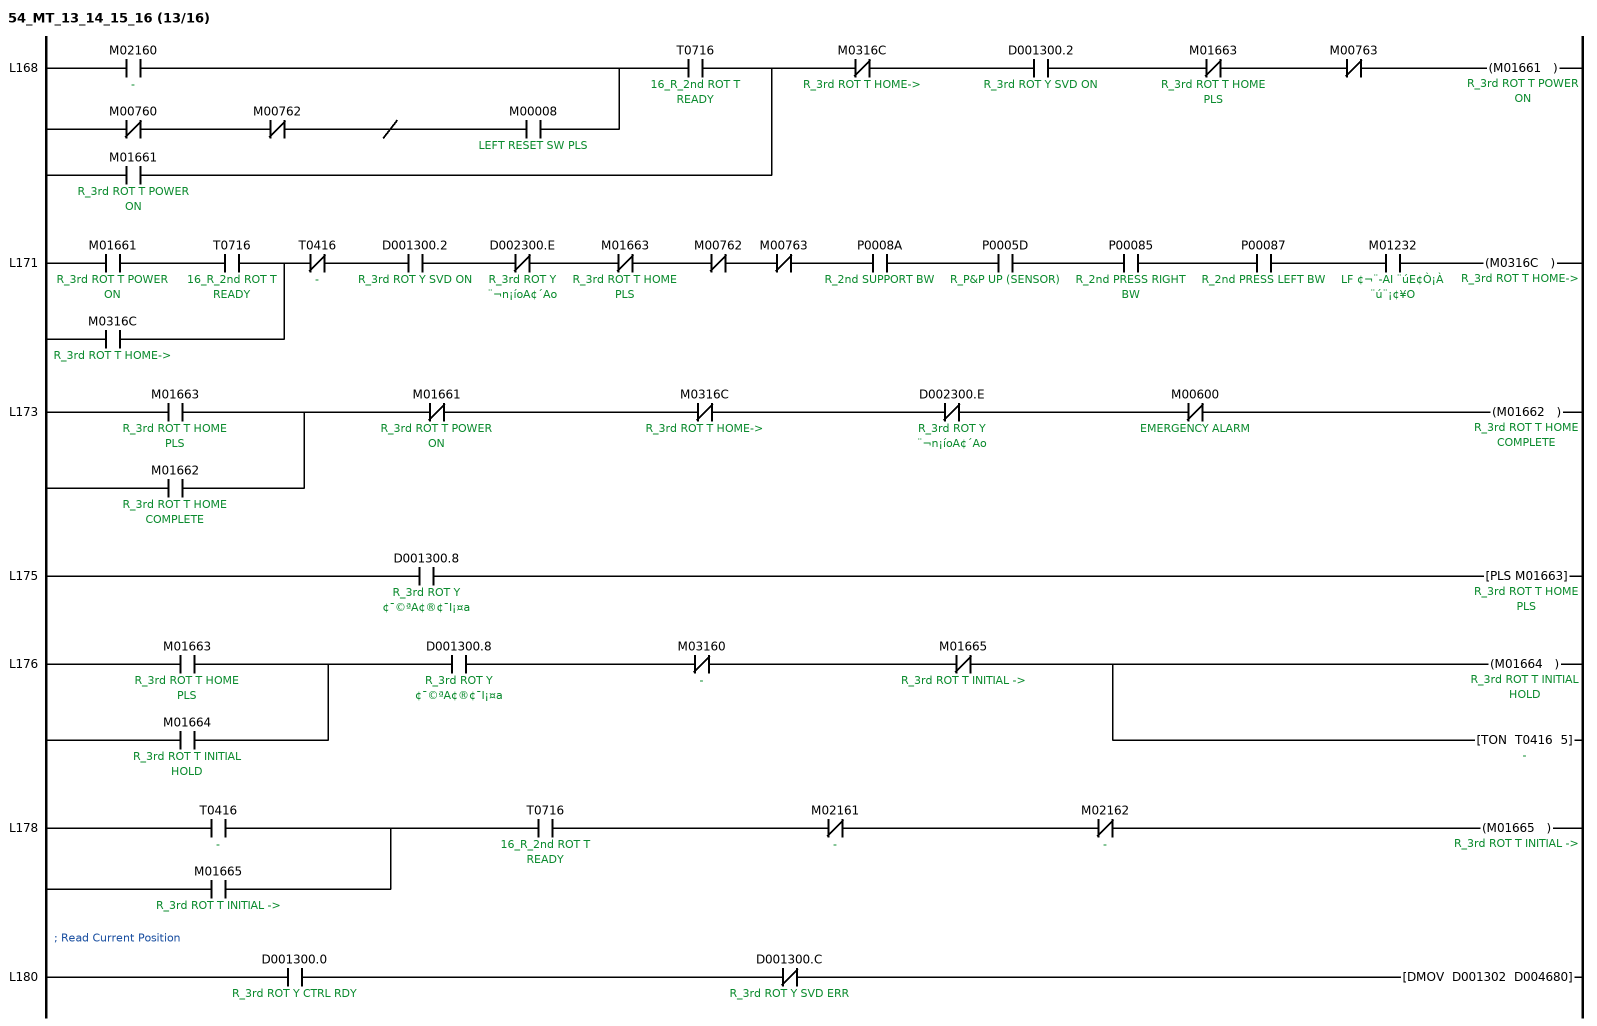
[picture p312: 54_MT_13_14_15_16 rungs L168-L180]
; L168
LOAD      M02160	// -
LOAD NOT  M00760
AND NOT   M00762
NOT
AND       M00008	// LEFT RESET SW PLS
OR LOAD
AND       T0716	// 16_R_2nd ROT T READY
OR        M01661	// R_3rd ROT T POWER ON
AND NOT   M0316C	// R_3rd ROT T HOME->
AND       D001300.2	// R_3rd ROT Y SVD ON
AND NOT   M01663	// R_3rd ROT T HOME PLS
AND NOT   M00763
OUT       M01661	// R_3rd ROT T POWER ON
; L171
LOAD      M01661	// R_3rd ROT T POWER ON
AND       T0716	// 16_R_2nd ROT T READY
OR        M0316C	// R_3rd ROT T HOME->
AND NOT   T0416	// -
AND       D001300.2	// R_3rd ROT Y SVD ON
AND NOT   D002300.E	// R_3rd ROT Y ¨¬n¡íoA¢´Ao
AND NOT   M01663	// R_3rd ROT T HOME PLS
AND NOT   M00762
AND NOT   M00763
AND       P0008A	// R_2nd SUPPORT BW
AND       P0005D	// R_P&P UP (SENSOR)
AND       P00085	// R_2nd PRESS RIGHT BW
AND       P00087	// R_2nd PRESS LEFT BW
AND       M01232	// LF ¢¬¨­AI ¨úE¢Ò¡À ¨ú¨¡¢¥O
OUT       M0316C	// R_3rd ROT T HOME->
; L173
LOAD      M01663	// R_3rd ROT T HOME PLS
OR        M01662	// R_3rd ROT T HOME COMPLETE
AND NOT   M01661	// R_3rd ROT T POWER ON
AND NOT   M0316C	// R_3rd ROT T HOME->
AND NOT   D002300.E	// R_3rd ROT Y ¨¬n¡íoA¢´Ao
AND NOT   M00600	// EMERGENCY ALARM
OUT       M01662	// R_3rd ROT T HOME COMPLETE
; L175
LOAD      D001300.8	// R_3rd ROT Y ¢¯©ªA¢®¢¯I¡¤a
OUTP      M01663	// R_3rd ROT T HOME PLS
; L176
LOAD      M01663	// R_3rd ROT T HOME PLS
OR        M01664	// R_3rd ROT T INITIAL HOLD
AND       D001300.8	// R_3rd ROT Y ¢¯©ªA¢®¢¯I¡¤a
AND NOT   M03160	// -
AND NOT   M01665	// R_3rd ROT T INITIAL ->
OUT       M01664	// R_3rd ROT T INITIAL HOLD
TON       T0416 5	// -
; L178
LOAD      T0416	// -
OR        M01665	// R_3rd ROT T INITIAL ->
AND       T0716	// 16_R_2nd ROT T READY
AND NOT   M02161	// -
AND NOT   M02162	// -
OUT       M01665	// R_3rd ROT T INITIAL ->
; L180
LOAD      D001300.0	// R_3rd ROT Y CTRL RDY
AND NOT   D001300.C	// R_3rd ROT Y SVD ERR
DMOV      D001302 D004680
// output comment: Read Current Position

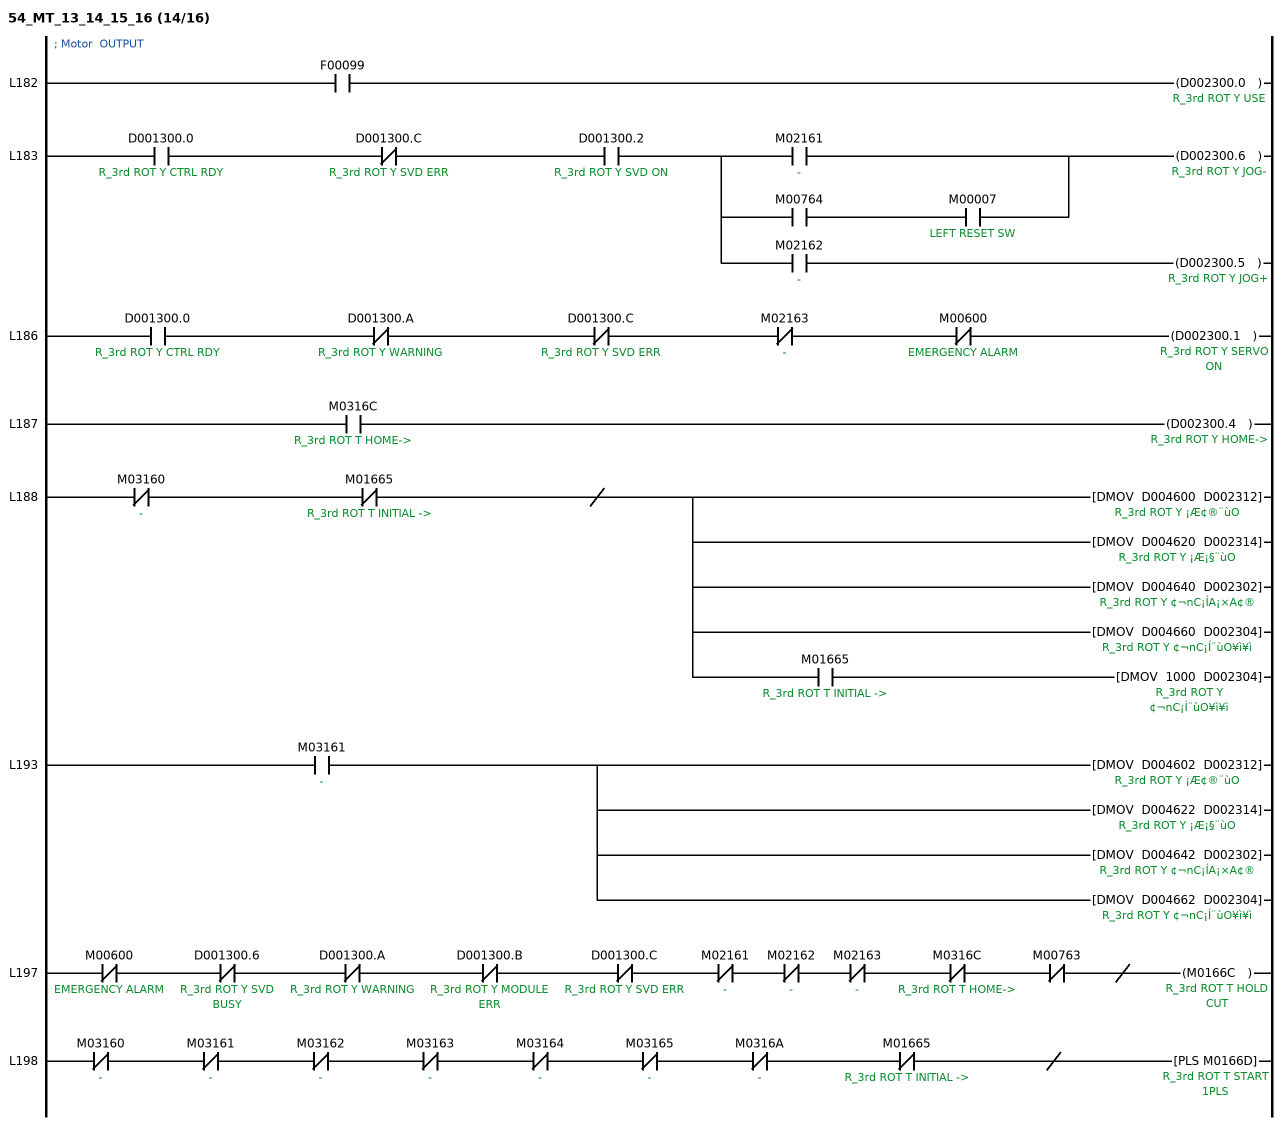
//  Motor  OUTPUT
; L182
LOAD      F00099
OUT       D002300.0	// R_3rd ROT Y USE
; L183
LOAD      D001300.0	// R_3rd ROT Y CTRL RDY
AND NOT   D001300.C	// R_3rd ROT Y SVD ERR
AND       D001300.2	// R_3rd ROT Y SVD ON
MPUSH
LOAD      M02161	// -
LOAD      M00764
AND       M00007	// LEFT RESET SW
OR LOAD
AND LOAD
OUT       D002300.6	// R_3rd ROT Y JOG-
MPOP
AND       M02162	// -
OUT       D002300.5	// R_3rd ROT Y JOG+
; L186
LOAD      D001300.0	// R_3rd ROT Y CTRL RDY
AND NOT   D001300.A	// R_3rd ROT Y WARNING
AND NOT   D001300.C	// R_3rd ROT Y SVD ERR
AND NOT   M02163	// -
AND NOT   M00600	// EMERGENCY ALARM
OUT       D002300.1	// R_3rd ROT Y SERVO ON
; L187
LOAD      M0316C	// R_3rd ROT T HOME->
OUT       D002300.4	// R_3rd ROT Y HOME->
; L188
LOAD NOT  M03160	// -
AND NOT   M01665	// R_3rd ROT T INITIAL ->
NOT
DMOV      D004600 D002312	// R_3rd ROT Y ¡Æ¢®¨ùO
DMOV      D004620 D002314	// R_3rd ROT Y ¡Æ¡§¨ùO
DMOV      D004640 D002302	// R_3rd ROT Y ¢¬nC¡ÍA¡×A¢®
DMOV      D004660 D002304	// R_3rd ROT Y ¢¬nC¡Í¨ùO¥ì¥ì
AND       M01665	// R_3rd ROT T INITIAL ->
DMOV      1000 D002304	// R_3rd ROT Y ¢¬nC¡Í¨ùO¥ì¥ì
; L193
LOAD      M03161	// -
DMOV      D004602 D002312	// R_3rd ROT Y ¡Æ¢®¨ùO
DMOV      D004622 D002314	// R_3rd ROT Y ¡Æ¡§¨ùO
DMOV      D004642 D002302	// R_3rd ROT Y ¢¬nC¡ÍA¡×A¢®
DMOV      D004662 D002304	// R_3rd ROT Y ¢¬nC¡Í¨ùO¥ì¥ì
; L197
LOAD NOT  M00600	// EMERGENCY ALARM
AND NOT   D001300.6	// R_3rd ROT Y SVD BUSY
AND NOT   D001300.A	// R_3rd ROT Y WARNING
AND NOT   D001300.B	// R_3rd ROT Y MODULE ERR
AND NOT   D001300.C	// R_3rd ROT Y SVD ERR
AND NOT   M02161	// -
AND NOT   M02162	// -
AND NOT   M02163	// -
AND NOT   M0316C	// R_3rd ROT T HOME->
AND NOT   M00763
NOT
OUT       M0166C	// R_3rd ROT T HOLD CUT
; L198
LOAD NOT  M03160	// -
AND NOT   M03161	// -
AND NOT   M03162	// -
AND NOT   M03163	// -
AND NOT   M03164	// -
AND NOT   M03165	// -
AND NOT   M0316A	// -
AND NOT   M01665	// R_3rd ROT T INITIAL ->
NOT
OUTP      M0166D	// R_3rd ROT T START 1PLS

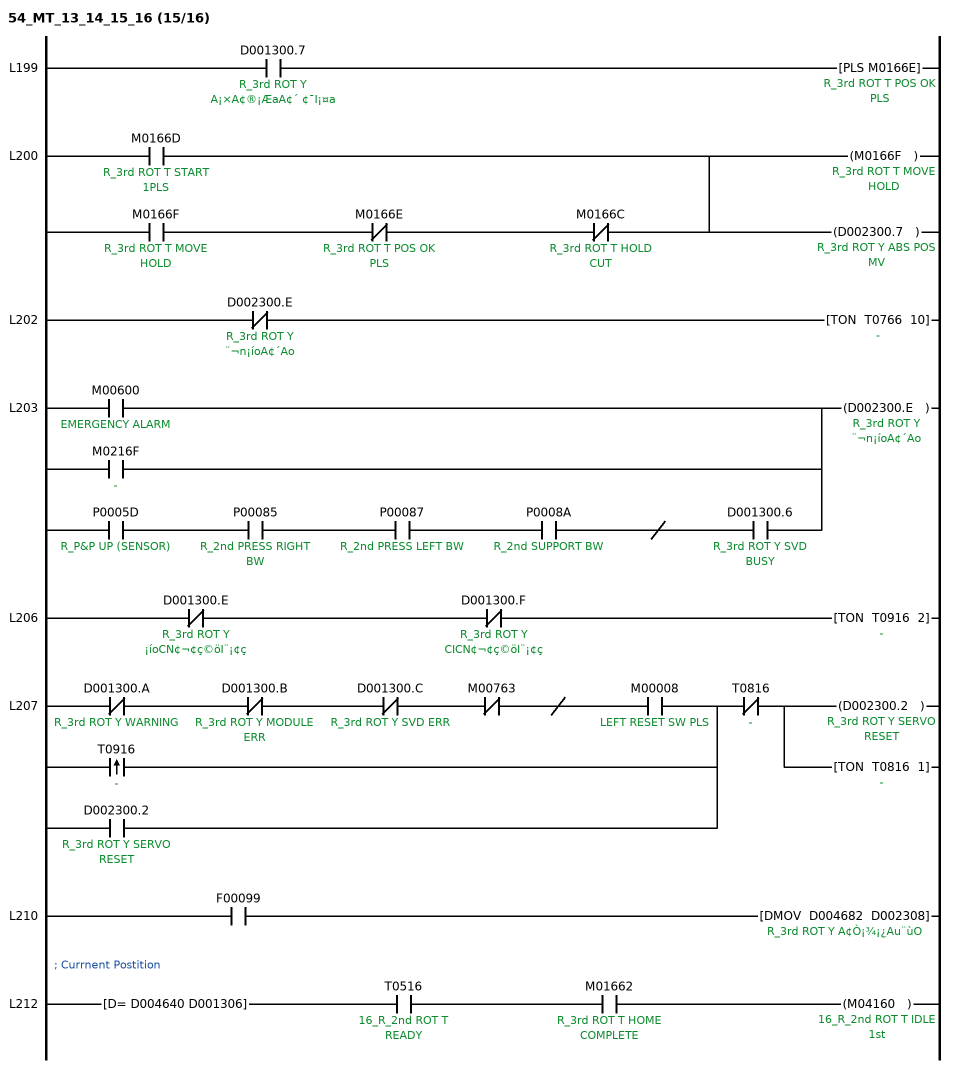
; L199
LOAD      D001300.7	// R_3rd ROT Y A¡×A¢®¡ÆaA¢´ ¢¯I¡¤a
OUTP      M0166E	// R_3rd ROT T POS OK PLS
; L200
LOAD      M0166D	// R_3rd ROT T START 1PLS
LOAD      M0166F	// R_3rd ROT T MOVE HOLD
AND NOT   M0166E	// R_3rd ROT T POS OK PLS
AND NOT   M0166C	// R_3rd ROT T HOLD CUT
OR LOAD
OUT       M0166F	// R_3rd ROT T MOVE HOLD
OUT       D002300.7	// R_3rd ROT Y ABS POS MV
; L202
LOAD NOT  D002300.E	// R_3rd ROT Y ¨¬n¡íoA¢´Ao
TON       T0766 10	// -
; L203
LOAD      M00600	// EMERGENCY ALARM
OR        M0216F	// -
LOAD      P0005D	// R_P&P UP (SENSOR)
AND       P00085	// R_2nd PRESS RIGHT BW
AND       P00087	// R_2nd PRESS LEFT BW
AND       P0008A	// R_2nd SUPPORT BW
NOT
AND       D001300.6	// R_3rd ROT Y SVD BUSY
OR LOAD
OUT       D002300.E	// R_3rd ROT Y ¨¬n¡íoA¢´Ao
; L206
LOAD NOT  D001300.E	// R_3rd ROT Y ¡íoCN¢¬¢ç©öI¨¡¢ç
AND NOT   D001300.F	// R_3rd ROT Y CICN¢¬¢ç©öI¨¡¢ç
TON       T0916 2	// -
; L207
LOAD NOT  D001300.A	// R_3rd ROT Y WARNING
AND NOT   D001300.B	// R_3rd ROT Y MODULE ERR
AND NOT   D001300.C	// R_3rd ROT Y SVD ERR
AND NOT   M00763
NOT
AND       M00008	// LEFT RESET SW PLS
ORP       T0916	// -
OR        D002300.2	// R_3rd ROT Y SERVO RESET
AND NOT   T0816	// -
OUT       D002300.2	// R_3rd ROT Y SERVO RESET
TON       T0816 1	// -
; L210
LOAD      F00099
DMOV      D004682 D002308	// R_3rd ROT Y A¢Ò¡¾¡¿Au¨ùO
// Currnent Postition
; L212
LOADD=    D004640 D001306
AND       T0516	// 16_R_2nd ROT T READY
AND       M01662	// R_3rd ROT T HOME COMPLETE
OUT       M04160	// 16_R_2nd ROT T IDLE 1st

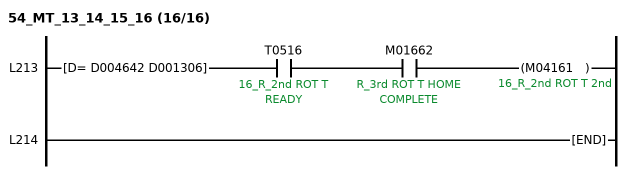
; L213
LOADD=    D004642 D001306
AND       T0516	// 16_R_2nd ROT T READY
AND       M01662	// R_3rd ROT T HOME COMPLETE
OUT       M04161	// 16_R_2nd ROT T 2nd
; L214
END

PROGRAM 55_MT_17_18_19_20 (task: ¨ö¨¬A¥ì CA¡¤I¡¾¡¿¡¤¡Í)

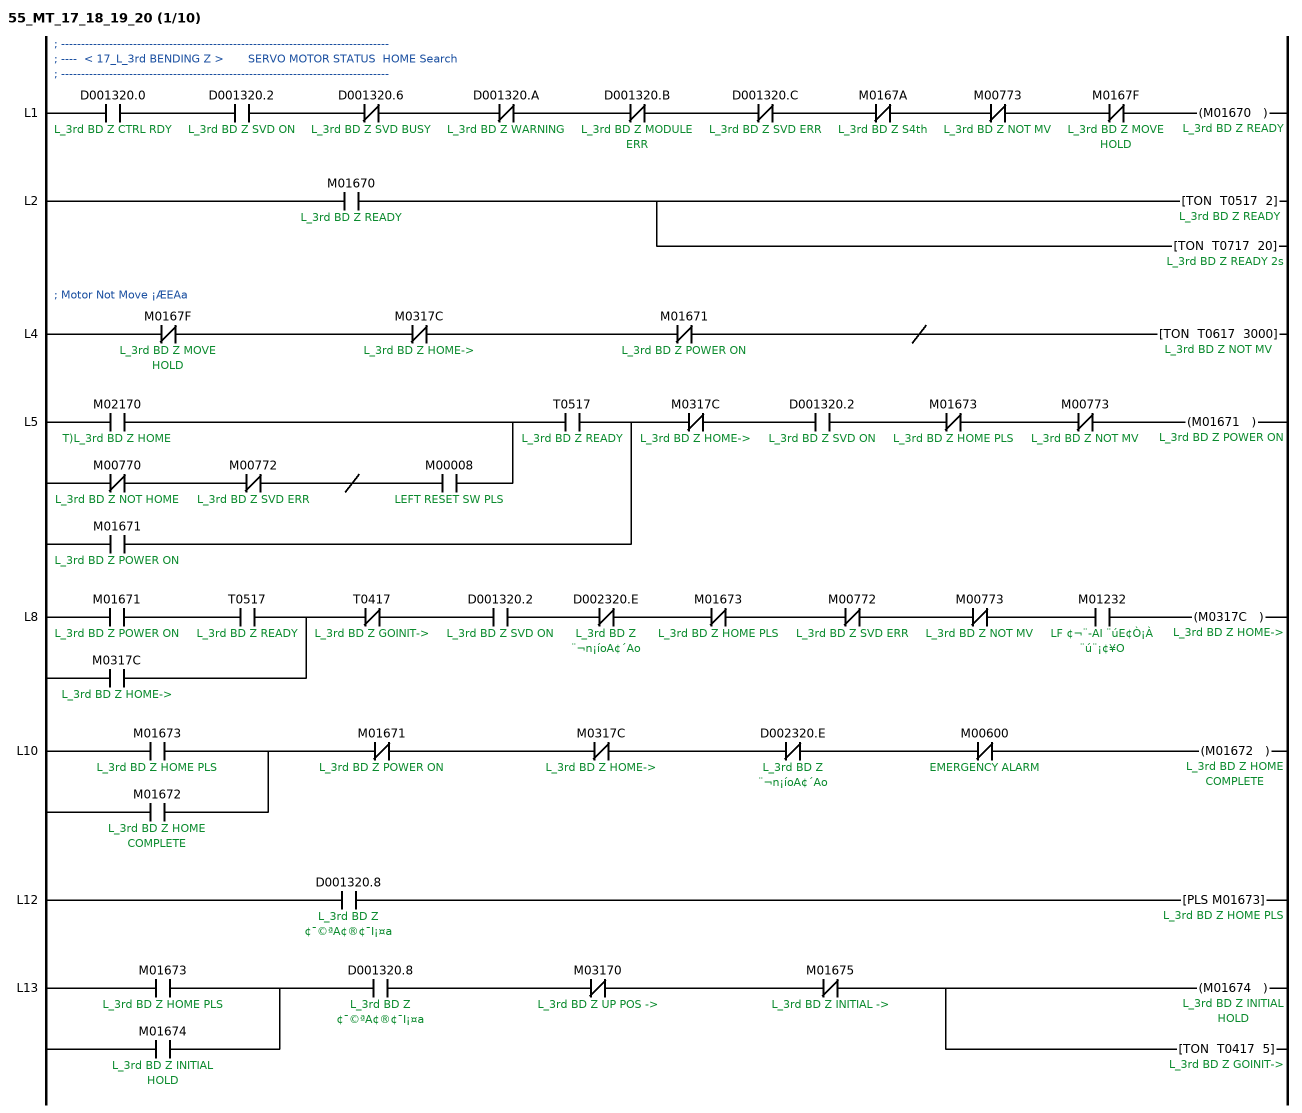
// ----------------------------------------------------------------------------------
// 
// ----  < 17_L_3rd BENDING Z >       SERVO MOTOR STATUS  HOME Search
// 
// ----------------------------------------------------------------------------------
; L1
LOAD      D001320.0	// L_3rd BD Z CTRL RDY
AND       D001320.2	// L_3rd BD Z SVD ON
AND NOT   D001320.6	// L_3rd BD Z SVD BUSY
AND NOT   D001320.A	// L_3rd BD Z WARNING
AND NOT   D001320.B	// L_3rd BD Z MODULE ERR
AND NOT   D001320.C	// L_3rd BD Z SVD ERR
AND NOT   M0167A	// L_3rd BD Z S4th
AND NOT   M00773	// L_3rd BD Z NOT MV
AND NOT   M0167F	// L_3rd BD Z MOVE HOLD
OUT       M01670	// L_3rd BD Z READY
; L2
LOAD      M01670	// L_3rd BD Z READY
TON       T0517 2	// L_3rd BD Z READY
TON       T0717 20	// L_3rd BD Z READY 2s
; L4
LOAD NOT  M0167F	// L_3rd BD Z MOVE HOLD
AND NOT   M0317C	// L_3rd BD Z HOME->
AND NOT   M01671	// L_3rd BD Z POWER ON
NOT
TON       T0617 3000	// L_3rd BD Z NOT MV
// output comment: Motor Not Move ¡ÆEAa
; L5
LOAD      M02170	// T)L_3rd BD Z HOME
LOAD NOT  M00770	// L_3rd BD Z NOT HOME
AND NOT   M00772	// L_3rd BD Z SVD ERR
NOT
AND       M00008	// LEFT RESET SW PLS
OR LOAD
AND       T0517	// L_3rd BD Z READY
OR        M01671	// L_3rd BD Z POWER ON
AND NOT   M0317C	// L_3rd BD Z HOME->
AND       D001320.2	// L_3rd BD Z SVD ON
AND NOT   M01673	// L_3rd BD Z HOME PLS
AND NOT   M00773	// L_3rd BD Z NOT MV
OUT       M01671	// L_3rd BD Z POWER ON
; L8
LOAD      M01671	// L_3rd BD Z POWER ON
AND       T0517	// L_3rd BD Z READY
OR        M0317C	// L_3rd BD Z HOME->
AND NOT   T0417	// L_3rd BD Z GOINIT->
AND       D001320.2	// L_3rd BD Z SVD ON
AND NOT   D002320.E	// L_3rd BD Z ¨¬n¡íoA¢´Ao
AND NOT   M01673	// L_3rd BD Z HOME PLS
AND NOT   M00772	// L_3rd BD Z SVD ERR
AND NOT   M00773	// L_3rd BD Z NOT MV
AND       M01232	// LF ¢¬¨­AI ¨úE¢Ò¡À ¨ú¨¡¢¥O
OUT       M0317C	// L_3rd BD Z HOME->
; L10
LOAD      M01673	// L_3rd BD Z HOME PLS
OR        M01672	// L_3rd BD Z HOME COMPLETE
AND NOT   M01671	// L_3rd BD Z POWER ON
AND NOT   M0317C	// L_3rd BD Z HOME->
AND NOT   D002320.E	// L_3rd BD Z ¨¬n¡íoA¢´Ao
AND NOT   M00600	// EMERGENCY ALARM
OUT       M01672	// L_3rd BD Z HOME COMPLETE
; L12
LOAD      D001320.8	// L_3rd BD Z ¢¯©ªA¢®¢¯I¡¤a
OUTP      M01673	// L_3rd BD Z HOME PLS
; L13
LOAD      M01673	// L_3rd BD Z HOME PLS
OR        M01674	// L_3rd BD Z INITIAL HOLD
AND       D001320.8	// L_3rd BD Z ¢¯©ªA¢®¢¯I¡¤a
AND NOT   M03170	// L_3rd BD Z UP POS ->
AND NOT   M01675	// L_3rd BD Z INITIAL ->
OUT       M01674	// L_3rd BD Z INITIAL HOLD
TON       T0417 5	// L_3rd BD Z GOINIT->

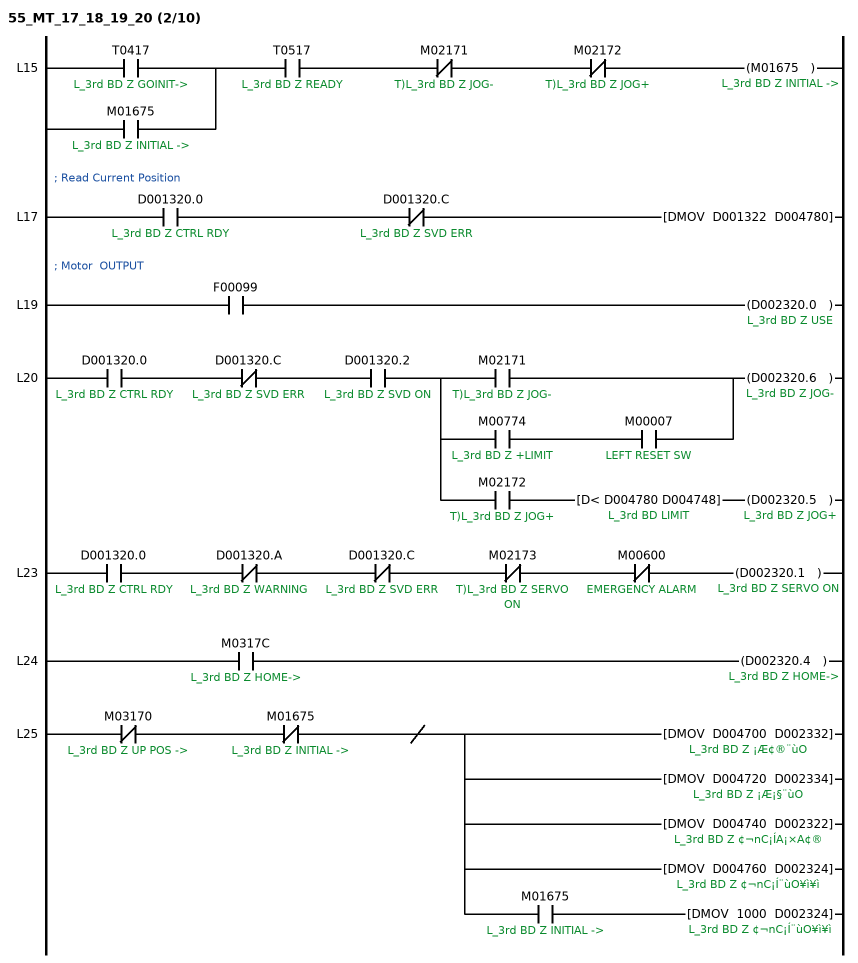
; L15
LOAD      T0417	// L_3rd BD Z GOINIT->
OR        M01675	// L_3rd BD Z INITIAL ->
AND       T0517	// L_3rd BD Z READY
AND NOT   M02171	// T)L_3rd BD Z JOG-
AND NOT   M02172	// T)L_3rd BD Z JOG+
OUT       M01675	// L_3rd BD Z INITIAL ->
; L17
LOAD      D001320.0	// L_3rd BD Z CTRL RDY
AND NOT   D001320.C	// L_3rd BD Z SVD ERR
DMOV      D001322 D004780
// output comment: Read Current Position
//  Motor  OUTPUT
; L19
LOAD      F00099
OUT       D002320.0	// L_3rd BD Z USE
; L20
LOAD      D001320.0	// L_3rd BD Z CTRL RDY
AND NOT   D001320.C	// L_3rd BD Z SVD ERR
AND       D001320.2	// L_3rd BD Z SVD ON
MPUSH
LOAD      M02171	// T)L_3rd BD Z JOG-
LOAD      M00774	// L_3rd BD Z +LIMIT
AND       M00007	// LEFT RESET SW
OR LOAD
AND LOAD
OUT       D002320.6	// L_3rd BD Z JOG-
MPOP
AND       M02172	// T)L_3rd BD Z JOG+
ANDD<     D004780 D004748	// L_3rd BD LIMIT
OUT       D002320.5	// L_3rd BD Z JOG+
; L23
LOAD      D001320.0	// L_3rd BD Z CTRL RDY
AND NOT   D001320.A	// L_3rd BD Z WARNING
AND NOT   D001320.C	// L_3rd BD Z SVD ERR
AND NOT   M02173	// T)L_3rd BD Z SERVO ON
AND NOT   M00600	// EMERGENCY ALARM
OUT       D002320.1	// L_3rd BD Z SERVO ON
; L24
LOAD      M0317C	// L_3rd BD Z HOME->
OUT       D002320.4	// L_3rd BD Z HOME->
; L25
LOAD NOT  M03170	// L_3rd BD Z UP POS ->
AND NOT   M01675	// L_3rd BD Z INITIAL ->
NOT
DMOV      D004700 D002332	// L_3rd BD Z ¡Æ¢®¨ùO
DMOV      D004720 D002334	// L_3rd BD Z ¡Æ¡§¨ùO
DMOV      D004740 D002322	// L_3rd BD Z ¢¬nC¡ÍA¡×A¢®
DMOV      D004760 D002324	// L_3rd BD Z ¢¬nC¡Í¨ùO¥ì¥ì
AND       M01675	// L_3rd BD Z INITIAL ->
DMOV      1000 D002324	// L_3rd BD Z ¢¬nC¡Í¨ùO¥ì¥ì

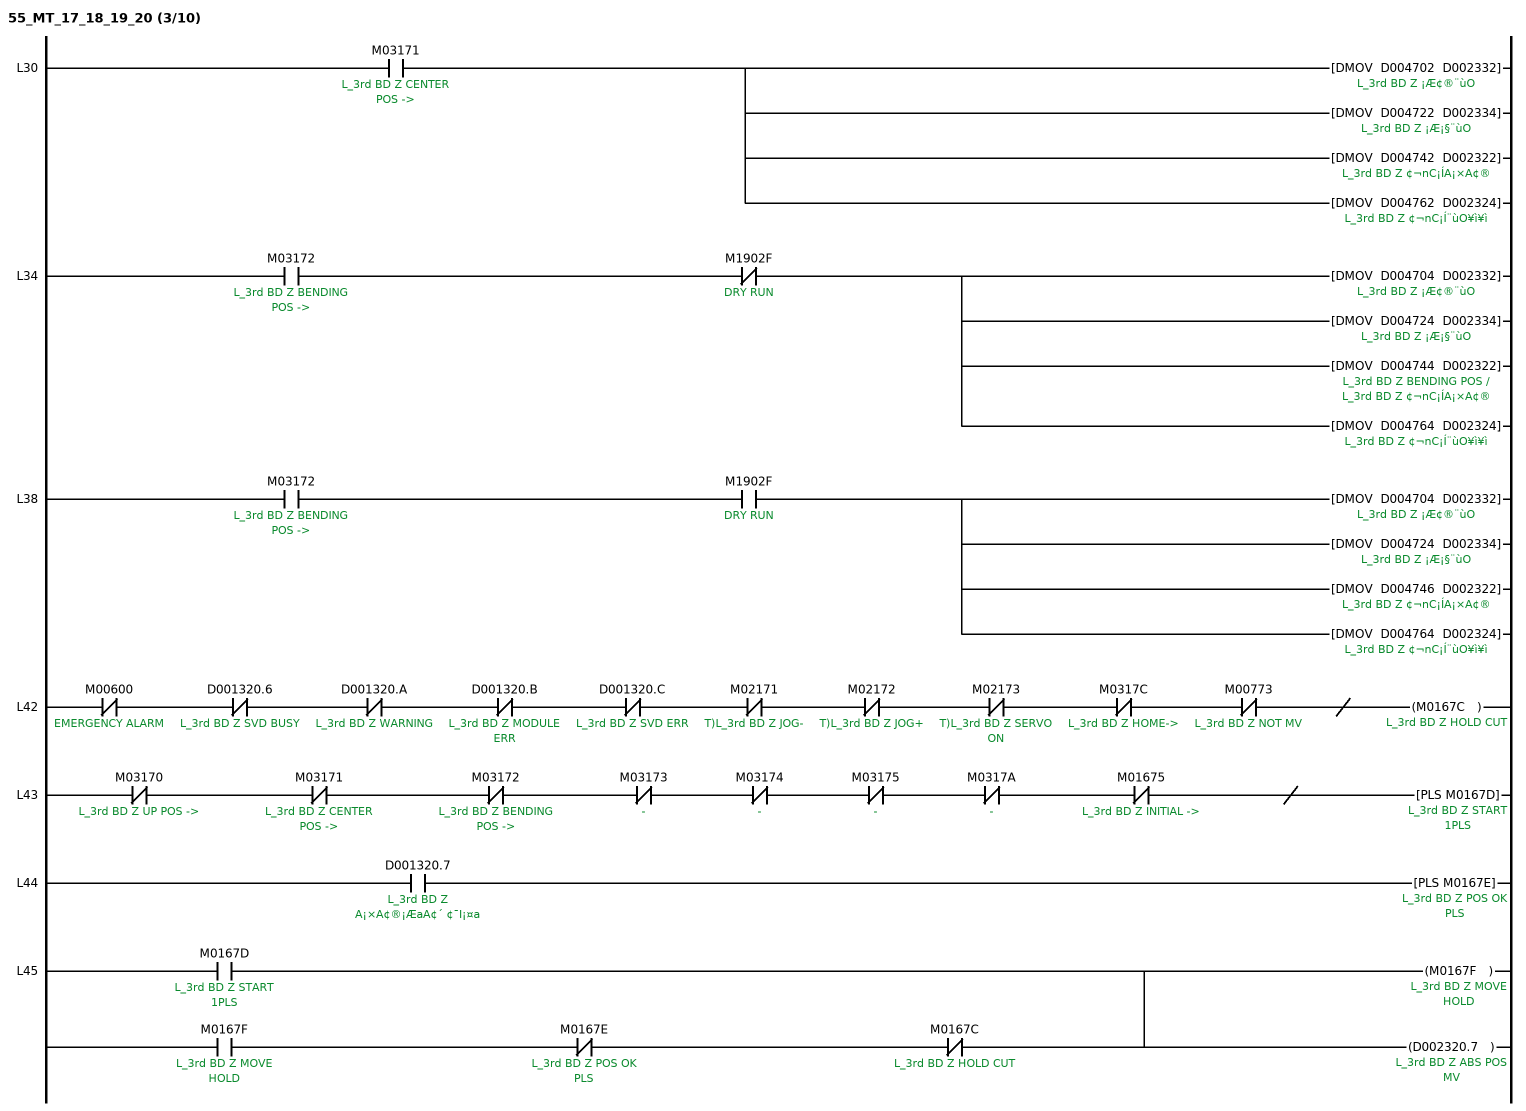
; L30
LOAD      M03171	// L_3rd BD Z CENTER POS ->
DMOV      D004702 D002332	// L_3rd BD Z ¡Æ¢®¨ùO
DMOV      D004722 D002334	// L_3rd BD Z ¡Æ¡§¨ùO
DMOV      D004742 D002322	// L_3rd BD Z ¢¬nC¡ÍA¡×A¢®
DMOV      D004762 D002324	// L_3rd BD Z ¢¬nC¡Í¨ùO¥ì¥ì
; L34
LOAD      M03172	// L_3rd BD Z BENDING POS ->
AND NOT   M1902F	// DRY RUN
DMOV      D004704 D002332	// L_3rd BD Z ¡Æ¢®¨ùO
DMOV      D004724 D002334	// L_3rd BD Z ¡Æ¡§¨ùO
DMOV      D004744 D002322	// L_3rd BD Z BENDING POS / L_3rd BD Z ¢¬nC¡ÍA¡×A¢®
DMOV      D004764 D002324	// L_3rd BD Z ¢¬nC¡Í¨ùO¥ì¥ì
; L38
LOAD      M03172	// L_3rd BD Z BENDING POS ->
AND       M1902F	// DRY RUN
DMOV      D004704 D002332	// L_3rd BD Z ¡Æ¢®¨ùO
DMOV      D004724 D002334	// L_3rd BD Z ¡Æ¡§¨ùO
DMOV      D004746 D002322	// L_3rd BD Z ¢¬nC¡ÍA¡×A¢®
DMOV      D004764 D002324	// L_3rd BD Z ¢¬nC¡Í¨ùO¥ì¥ì
; L42
LOAD NOT  M00600	// EMERGENCY ALARM
AND NOT   D001320.6	// L_3rd BD Z SVD BUSY
AND NOT   D001320.A	// L_3rd BD Z WARNING
AND NOT   D001320.B	// L_3rd BD Z MODULE ERR
AND NOT   D001320.C	// L_3rd BD Z SVD ERR
AND NOT   M02171	// T)L_3rd BD Z JOG-
AND NOT   M02172	// T)L_3rd BD Z JOG+
AND NOT   M02173	// T)L_3rd BD Z SERVO ON
AND NOT   M0317C	// L_3rd BD Z HOME->
AND NOT   M00773	// L_3rd BD Z NOT MV
NOT
OUT       M0167C	// L_3rd BD Z HOLD CUT
; L43
LOAD NOT  M03170	// L_3rd BD Z UP POS ->
AND NOT   M03171	// L_3rd BD Z CENTER POS ->
AND NOT   M03172	// L_3rd BD Z BENDING POS ->
AND NOT   M03173	// -
AND NOT   M03174	// -
AND NOT   M03175	// -
AND NOT   M0317A	// -
AND NOT   M01675	// L_3rd BD Z INITIAL ->
NOT
OUTP      M0167D	// L_3rd BD Z START 1PLS
; L44
LOAD      D001320.7	// L_3rd BD Z A¡×A¢®¡ÆaA¢´ ¢¯I¡¤a
OUTP      M0167E	// L_3rd BD Z POS OK PLS
; L45
LOAD      M0167D	// L_3rd BD Z START 1PLS
LOAD      M0167F	// L_3rd BD Z MOVE HOLD
AND NOT   M0167E	// L_3rd BD Z POS OK PLS
AND NOT   M0167C	// L_3rd BD Z HOLD CUT
OR LOAD
OUT       M0167F	// L_3rd BD Z MOVE HOLD
OUT       D002320.7	// L_3rd BD Z ABS POS MV

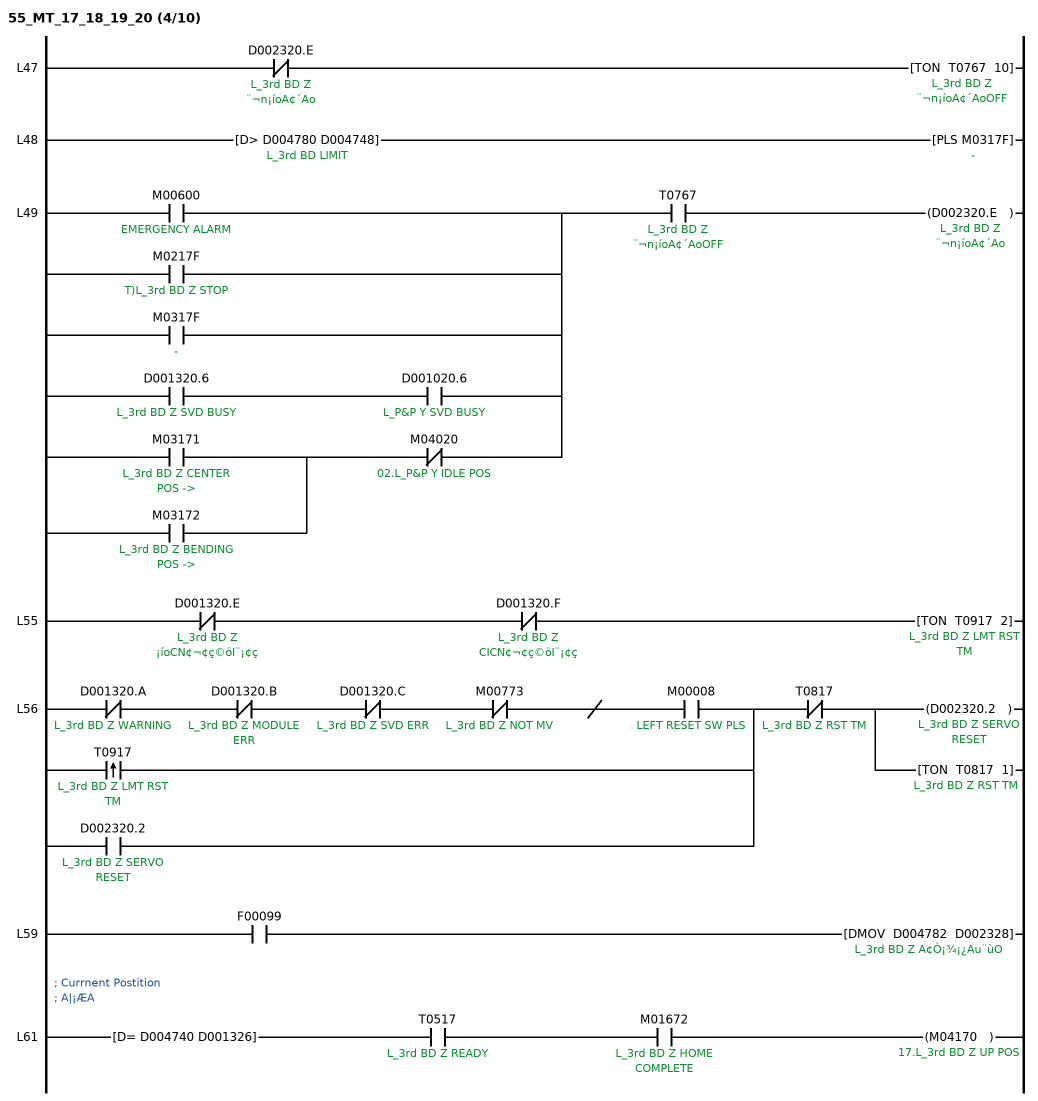
; L47
LOAD NOT  D002320.E	// L_3rd BD Z ¨¬n¡íoA¢´Ao
TON       T0767 10	// L_3rd BD Z ¨¬n¡íoA¢´AoOFF
; L48
LOADD>    D004780 D004748	// L_3rd BD LIMIT
OUTP      M0317F	// -
; L49
LOAD      M00600	// EMERGENCY ALARM
OR        M0217F	// T)L_3rd BD Z STOP
OR        M0317F	// -
LOAD      D001320.6	// L_3rd BD Z SVD BUSY
AND       D001020.6	// L_P&P Y SVD BUSY
OR LOAD
LOAD      M03171	// L_3rd BD Z CENTER POS ->
OR        M03172	// L_3rd BD Z BENDING POS ->
AND NOT   M04020	// 02.L_P&P Y IDLE POS
OR LOAD
AND       T0767	// L_3rd BD Z ¨¬n¡íoA¢´AoOFF
OUT       D002320.E	// L_3rd BD Z ¨¬n¡íoA¢´Ao
; L55
LOAD NOT  D001320.E	// L_3rd BD Z ¡íoCN¢¬¢ç©öI¨¡¢ç
AND NOT   D001320.F	// L_3rd BD Z CICN¢¬¢ç©öI¨¡¢ç
TON       T0917 2	// L_3rd BD Z LMT RST TM
; L56
LOAD NOT  D001320.A	// L_3rd BD Z WARNING
AND NOT   D001320.B	// L_3rd BD Z MODULE ERR
AND NOT   D001320.C	// L_3rd BD Z SVD ERR
AND NOT   M00773	// L_3rd BD Z NOT MV
NOT
AND       M00008	// LEFT RESET SW PLS
ORP       T0917	// L_3rd BD Z LMT RST TM
OR        D002320.2	// L_3rd BD Z SERVO RESET
AND NOT   T0817	// L_3rd BD Z RST TM
OUT       D002320.2	// L_3rd BD Z SERVO RESET
TON       T0817 1	// L_3rd BD Z RST TM
; L59
LOAD      F00099
DMOV      D004782 D002328	// L_3rd BD Z A¢Ò¡¾¡¿Au¨ùO
// Currnent Postition
; L61
LOADD=    D004740 D001326
AND       T0517	// L_3rd BD Z READY
AND       M01672	// L_3rd BD Z HOME COMPLETE
OUT       M04170	// 17.L_3rd BD Z UP POS
// output comment: A|¡ÆA

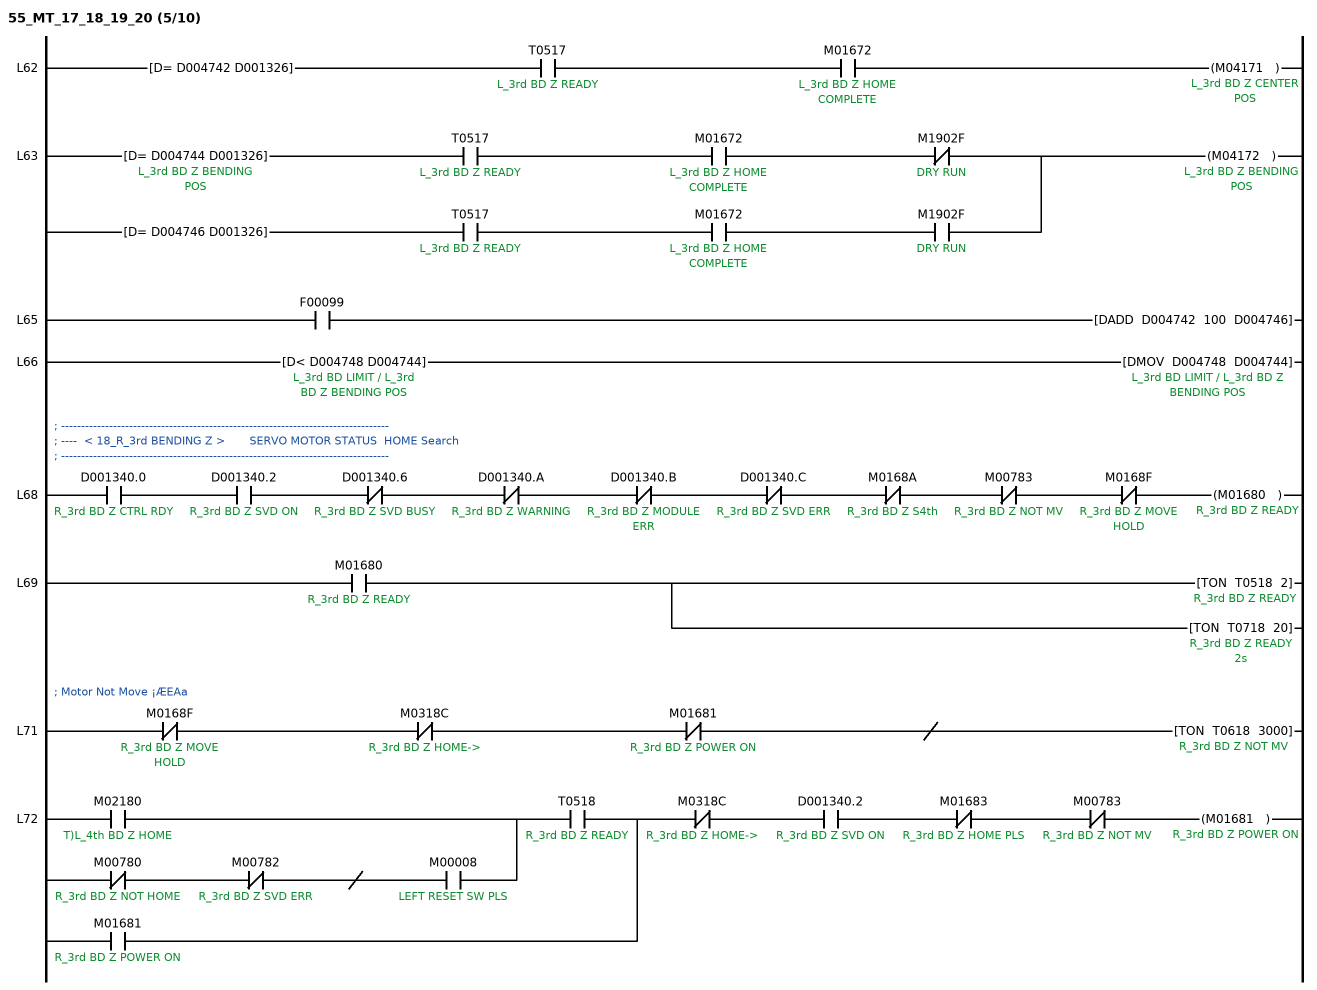
; L62
LOADD=    D004742 D001326
AND       T0517	// L_3rd BD Z READY
AND       M01672	// L_3rd BD Z HOME COMPLETE
OUT       M04171	// L_3rd BD Z CENTER POS
; L63
LOADD=    D004744 D001326	// L_3rd BD Z BENDING POS
AND       T0517	// L_3rd BD Z READY
AND       M01672	// L_3rd BD Z HOME COMPLETE
AND NOT   M1902F	// DRY RUN
LOADD=    D004746 D001326
AND       T0517	// L_3rd BD Z READY
AND       M01672	// L_3rd BD Z HOME COMPLETE
AND       M1902F	// DRY RUN
OR LOAD
OUT       M04172	// L_3rd BD Z BENDING POS
; L65
LOAD      F00099
DADD      D004742 100 D004746
; L66
LOADD<    D004748 D004744	// L_3rd BD LIMIT / L_3rd BD Z BENDING POS
DMOV      D004748 D004744	// L_3rd BD LIMIT / L_3rd BD Z BENDING POS
// ----------------------------------------------------------------------------------
// 
// ----  < 18_R_3rd BENDING Z >       SERVO MOTOR STATUS  HOME Search
// 
// ----------------------------------------------------------------------------------
; L68
LOAD      D001340.0	// R_3rd BD Z CTRL RDY
AND       D001340.2	// R_3rd BD Z SVD ON
AND NOT   D001340.6	// R_3rd BD Z SVD BUSY
AND NOT   D001340.A	// R_3rd BD Z WARNING
AND NOT   D001340.B	// R_3rd BD Z MODULE ERR
AND NOT   D001340.C	// R_3rd BD Z SVD ERR
AND NOT   M0168A	// R_3rd BD Z S4th
AND NOT   M00783	// R_3rd BD Z NOT MV
AND NOT   M0168F	// R_3rd BD Z MOVE HOLD
OUT       M01680	// R_3rd BD Z READY
; L69
LOAD      M01680	// R_3rd BD Z READY
TON       T0518 2	// R_3rd BD Z READY
TON       T0718 20	// R_3rd BD Z READY 2s
; L71
LOAD NOT  M0168F	// R_3rd BD Z MOVE HOLD
AND NOT   M0318C	// R_3rd BD Z HOME->
AND NOT   M01681	// R_3rd BD Z POWER ON
NOT
TON       T0618 3000	// R_3rd BD Z NOT MV
// output comment: Motor Not Move ¡ÆEAa
; L72
LOAD      M02180	// T)L_4th BD Z HOME
LOAD NOT  M00780	// R_3rd BD Z NOT HOME
AND NOT   M00782	// R_3rd BD Z SVD ERR
NOT
AND       M00008	// LEFT RESET SW PLS
OR LOAD
AND       T0518	// R_3rd BD Z READY
OR        M01681	// R_3rd BD Z POWER ON
AND NOT   M0318C	// R_3rd BD Z HOME->
AND       D001340.2	// R_3rd BD Z SVD ON
AND NOT   M01683	// R_3rd BD Z HOME PLS
AND NOT   M00783	// R_3rd BD Z NOT MV
OUT       M01681	// R_3rd BD Z POWER ON

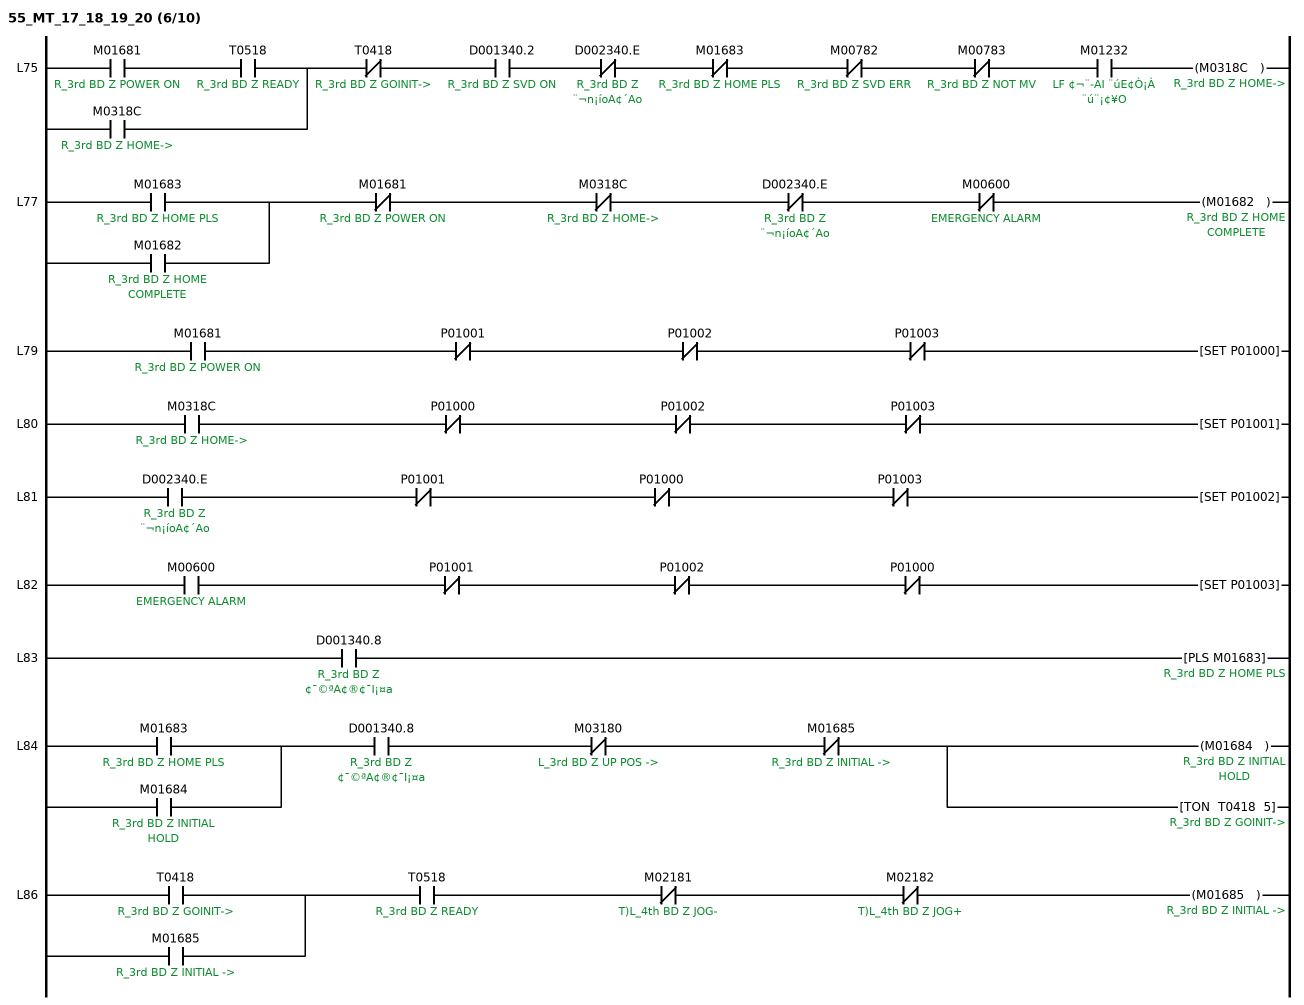
; L75
LOAD      M01681	// R_3rd BD Z POWER ON
AND       T0518	// R_3rd BD Z READY
OR        M0318C	// R_3rd BD Z HOME->
AND NOT   T0418	// R_3rd BD Z GOINIT->
AND       D001340.2	// R_3rd BD Z SVD ON
AND NOT   D002340.E	// R_3rd BD Z ¨¬n¡íoA¢´Ao
AND NOT   M01683	// R_3rd BD Z HOME PLS
AND NOT   M00782	// R_3rd BD Z SVD ERR
AND NOT   M00783	// R_3rd BD Z NOT MV
AND       M01232	// LF ¢¬¨­AI ¨úE¢Ò¡À ¨ú¨¡¢¥O
OUT       M0318C	// R_3rd BD Z HOME->
; L77
LOAD      M01683	// R_3rd BD Z HOME PLS
OR        M01682	// R_3rd BD Z HOME COMPLETE
AND NOT   M01681	// R_3rd BD Z POWER ON
AND NOT   M0318C	// R_3rd BD Z HOME->
AND NOT   D002340.E	// R_3rd BD Z ¨¬n¡íoA¢´Ao
AND NOT   M00600	// EMERGENCY ALARM
OUT       M01682	// R_3rd BD Z HOME COMPLETE
; L79
LOAD      M01681	// R_3rd BD Z POWER ON
AND NOT   P01001
AND NOT   P01002
AND NOT   P01003
SET       P01000
; L80
LOAD      M0318C	// R_3rd BD Z HOME->
AND NOT   P01000
AND NOT   P01002
AND NOT   P01003
SET       P01001
; L81
LOAD      D002340.E	// R_3rd BD Z ¨¬n¡íoA¢´Ao
AND NOT   P01001
AND NOT   P01000
AND NOT   P01003
SET       P01002
; L82
LOAD      M00600	// EMERGENCY ALARM
AND NOT   P01001
AND NOT   P01002
AND NOT   P01000
SET       P01003
; L83
LOAD      D001340.8	// R_3rd BD Z ¢¯©ªA¢®¢¯I¡¤a
OUTP      M01683	// R_3rd BD Z HOME PLS
; L84
LOAD      M01683	// R_3rd BD Z HOME PLS
OR        M01684	// R_3rd BD Z INITIAL HOLD
AND       D001340.8	// R_3rd BD Z ¢¯©ªA¢®¢¯I¡¤a
AND NOT   M03180	// L_3rd BD Z UP POS ->
AND NOT   M01685	// R_3rd BD Z INITIAL ->
OUT       M01684	// R_3rd BD Z INITIAL HOLD
TON       T0418 5	// R_3rd BD Z GOINIT->
; L86
LOAD      T0418	// R_3rd BD Z GOINIT->
OR        M01685	// R_3rd BD Z INITIAL ->
AND       T0518	// R_3rd BD Z READY
AND NOT   M02181	// T)L_4th BD Z JOG-
AND NOT   M02182	// T)L_4th BD Z JOG+
OUT       M01685	// R_3rd BD Z INITIAL ->

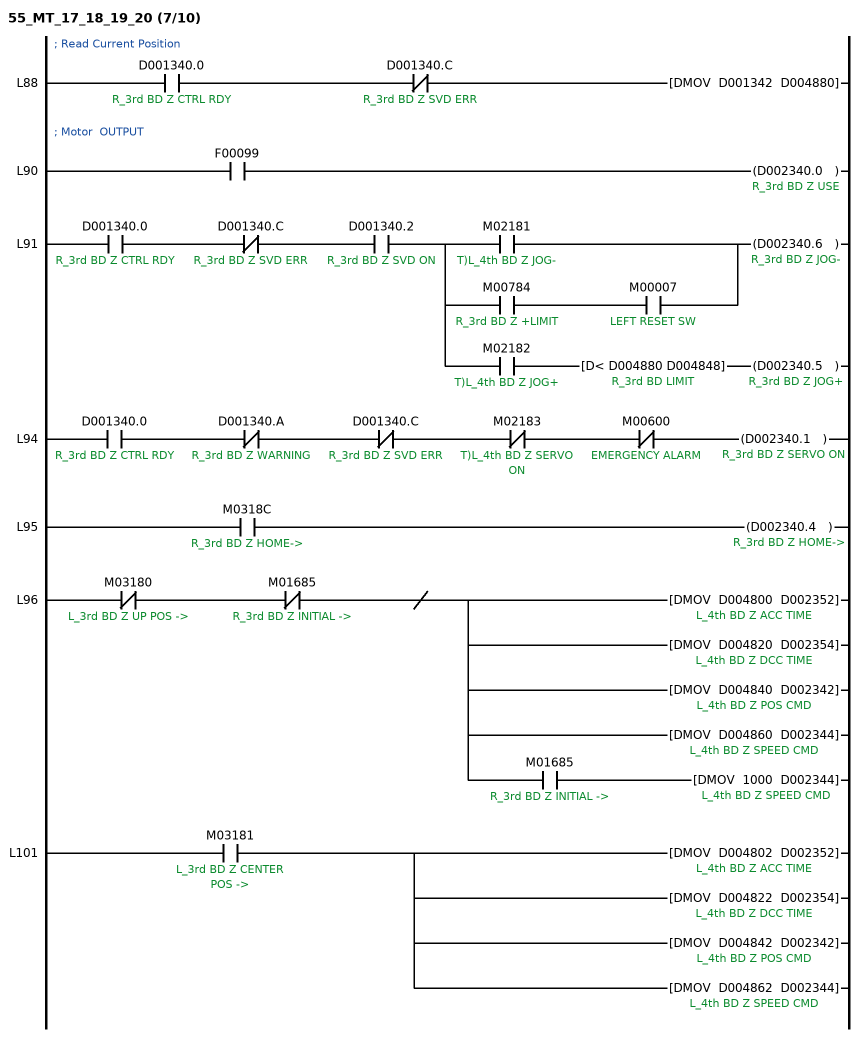
; L88
LOAD      D001340.0	// R_3rd BD Z CTRL RDY
AND NOT   D001340.C	// R_3rd BD Z SVD ERR
DMOV      D001342 D004880
// output comment: Read Current Position
//  Motor  OUTPUT
; L90
LOAD      F00099
OUT       D002340.0	// R_3rd BD Z USE
; L91
LOAD      D001340.0	// R_3rd BD Z CTRL RDY
AND NOT   D001340.C	// R_3rd BD Z SVD ERR
AND       D001340.2	// R_3rd BD Z SVD ON
MPUSH
LOAD      M02181	// T)L_4th BD Z JOG-
LOAD      M00784	// R_3rd BD Z +LIMIT
AND       M00007	// LEFT RESET SW
OR LOAD
AND LOAD
OUT       D002340.6	// R_3rd BD Z JOG-
MPOP
AND       M02182	// T)L_4th BD Z JOG+
ANDD<     D004880 D004848	// R_3rd BD LIMIT
OUT       D002340.5	// R_3rd BD Z JOG+
; L94
LOAD      D001340.0	// R_3rd BD Z CTRL RDY
AND NOT   D001340.A	// R_3rd BD Z WARNING
AND NOT   D001340.C	// R_3rd BD Z SVD ERR
AND NOT   M02183	// T)L_4th BD Z SERVO ON
AND NOT   M00600	// EMERGENCY ALARM
OUT       D002340.1	// R_3rd BD Z SERVO ON
; L95
LOAD      M0318C	// R_3rd BD Z HOME->
OUT       D002340.4	// R_3rd BD Z HOME->
; L96
LOAD NOT  M03180	// L_3rd BD Z UP POS ->
AND NOT   M01685	// R_3rd BD Z INITIAL ->
NOT
DMOV      D004800 D002352	// L_4th BD Z ACC TIME
DMOV      D004820 D002354	// L_4th BD Z DCC TIME
DMOV      D004840 D002342	// L_4th BD Z POS CMD
DMOV      D004860 D002344	// L_4th BD Z SPEED CMD
AND       M01685	// R_3rd BD Z INITIAL ->
DMOV      1000 D002344	// L_4th BD Z SPEED CMD
; L101
LOAD      M03181	// L_3rd BD Z CENTER POS ->
DMOV      D004802 D002352	// L_4th BD Z ACC TIME
DMOV      D004822 D002354	// L_4th BD Z DCC TIME
DMOV      D004842 D002342	// L_4th BD Z POS CMD
DMOV      D004862 D002344	// L_4th BD Z SPEED CMD

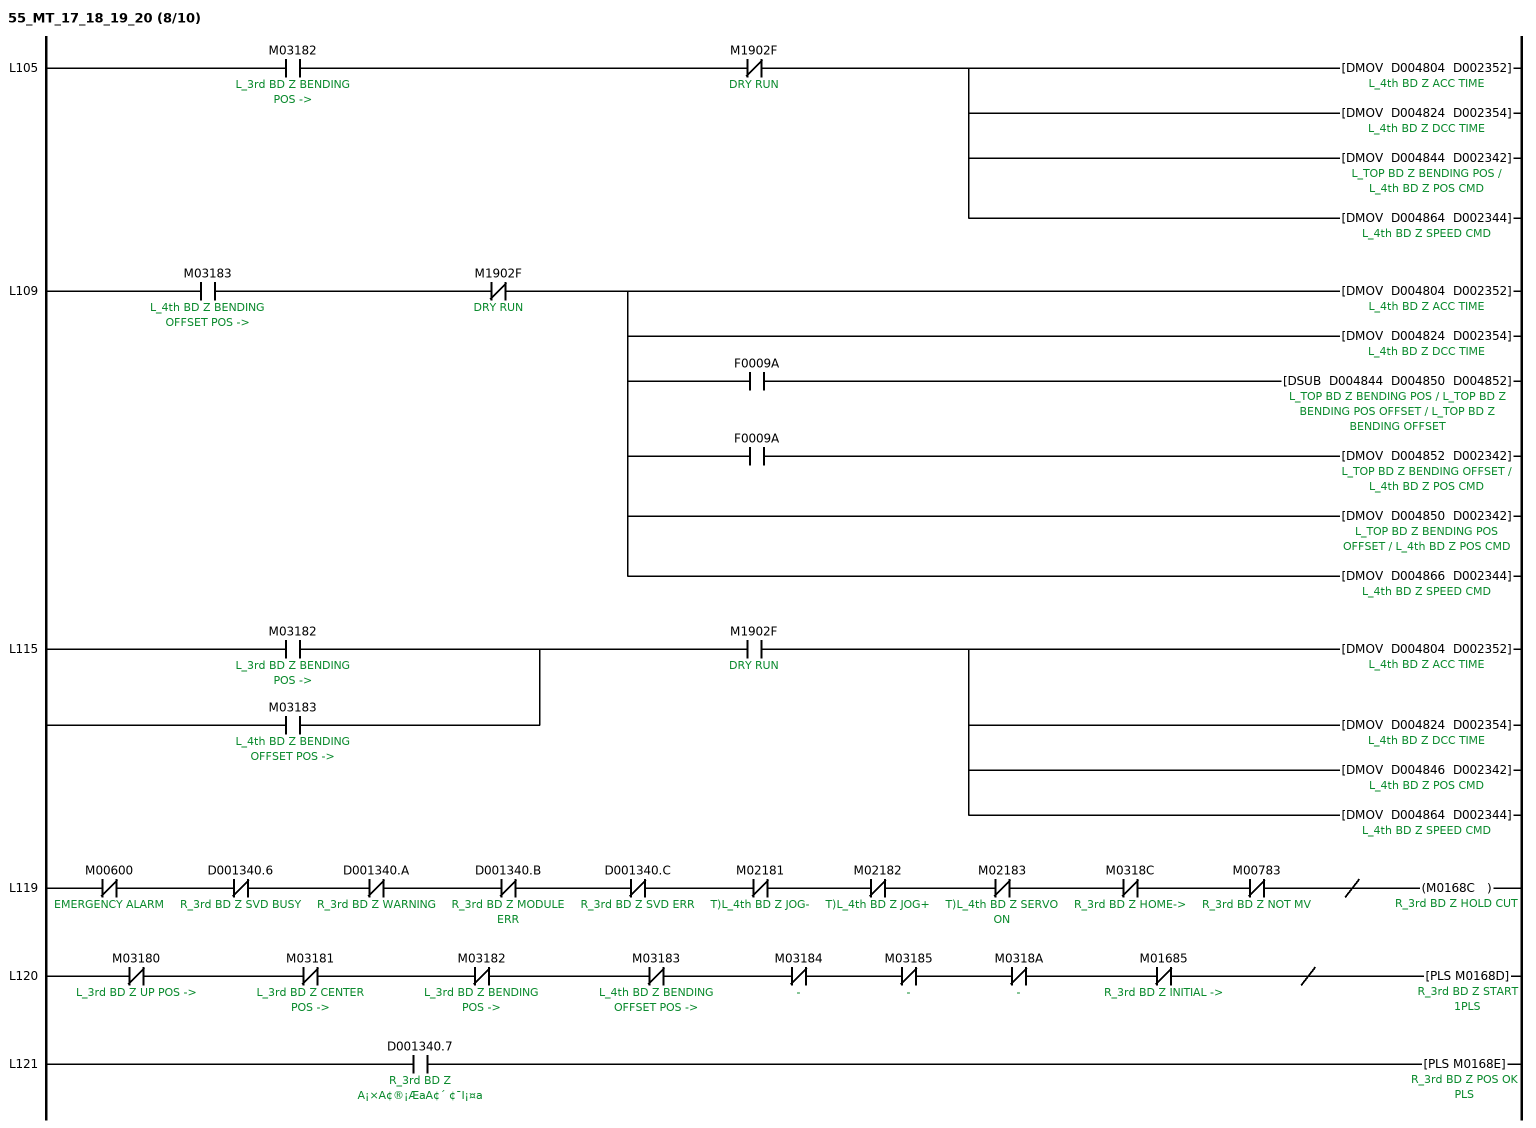
; L105
LOAD      M03182	// L_3rd BD Z BENDING POS ->
AND NOT   M1902F	// DRY RUN
DMOV      D004804 D002352	// L_4th BD Z ACC TIME
DMOV      D004824 D002354	// L_4th BD Z DCC TIME
DMOV      D004844 D002342	// L_TOP BD Z BENDING POS / L_4th BD Z POS CMD
DMOV      D004864 D002344	// L_4th BD Z SPEED CMD
; L109
LOAD      M03183	// L_4th BD Z BENDING OFFSET POS ->
AND NOT   M1902F	// DRY RUN
DMOV      D004804 D002352	// L_4th BD Z ACC TIME
DMOV      D004824 D002354	// L_4th BD Z DCC TIME
MPUSH
AND       F0009A
DSUB      D004844 D004850 D004852	// L_TOP BD Z BENDING POS / L_TOP BD Z BENDING POS OFFSET / L_TOP BD Z BENDING OFFSET
MLOAD
AND       F0009A
DMOV      D004852 D002342	// L_TOP BD Z BENDING OFFSET / L_4th BD Z POS CMD
MPOP
DMOV      D004850 D002342	// L_TOP BD Z BENDING POS OFFSET / L_4th BD Z POS CMD
DMOV      D004866 D002344	// L_4th BD Z SPEED CMD
; L115
LOAD      M03182	// L_3rd BD Z BENDING POS ->
OR        M03183	// L_4th BD Z BENDING OFFSET POS ->
AND       M1902F	// DRY RUN
DMOV      D004804 D002352	// L_4th BD Z ACC TIME
DMOV      D004824 D002354	// L_4th BD Z DCC TIME
DMOV      D004846 D002342	// L_4th BD Z POS CMD
DMOV      D004864 D002344	// L_4th BD Z SPEED CMD
; L119
LOAD NOT  M00600	// EMERGENCY ALARM
AND NOT   D001340.6	// R_3rd BD Z SVD BUSY
AND NOT   D001340.A	// R_3rd BD Z WARNING
AND NOT   D001340.B	// R_3rd BD Z MODULE ERR
AND NOT   D001340.C	// R_3rd BD Z SVD ERR
AND NOT   M02181	// T)L_4th BD Z JOG-
AND NOT   M02182	// T)L_4th BD Z JOG+
AND NOT   M02183	// T)L_4th BD Z SERVO ON
AND NOT   M0318C	// R_3rd BD Z HOME->
AND NOT   M00783	// R_3rd BD Z NOT MV
NOT
OUT       M0168C	// R_3rd BD Z HOLD CUT
; L120
LOAD NOT  M03180	// L_3rd BD Z UP POS ->
AND NOT   M03181	// L_3rd BD Z CENTER POS ->
AND NOT   M03182	// L_3rd BD Z BENDING POS ->
AND NOT   M03183	// L_4th BD Z BENDING OFFSET POS ->
AND NOT   M03184	// -
AND NOT   M03185	// -
AND NOT   M0318A	// -
AND NOT   M01685	// R_3rd BD Z INITIAL ->
NOT
OUTP      M0168D	// R_3rd BD Z START 1PLS
; L121
LOAD      D001340.7	// R_3rd BD Z A¡×A¢®¡ÆaA¢´ ¢¯I¡¤a
OUTP      M0168E	// R_3rd BD Z POS OK PLS

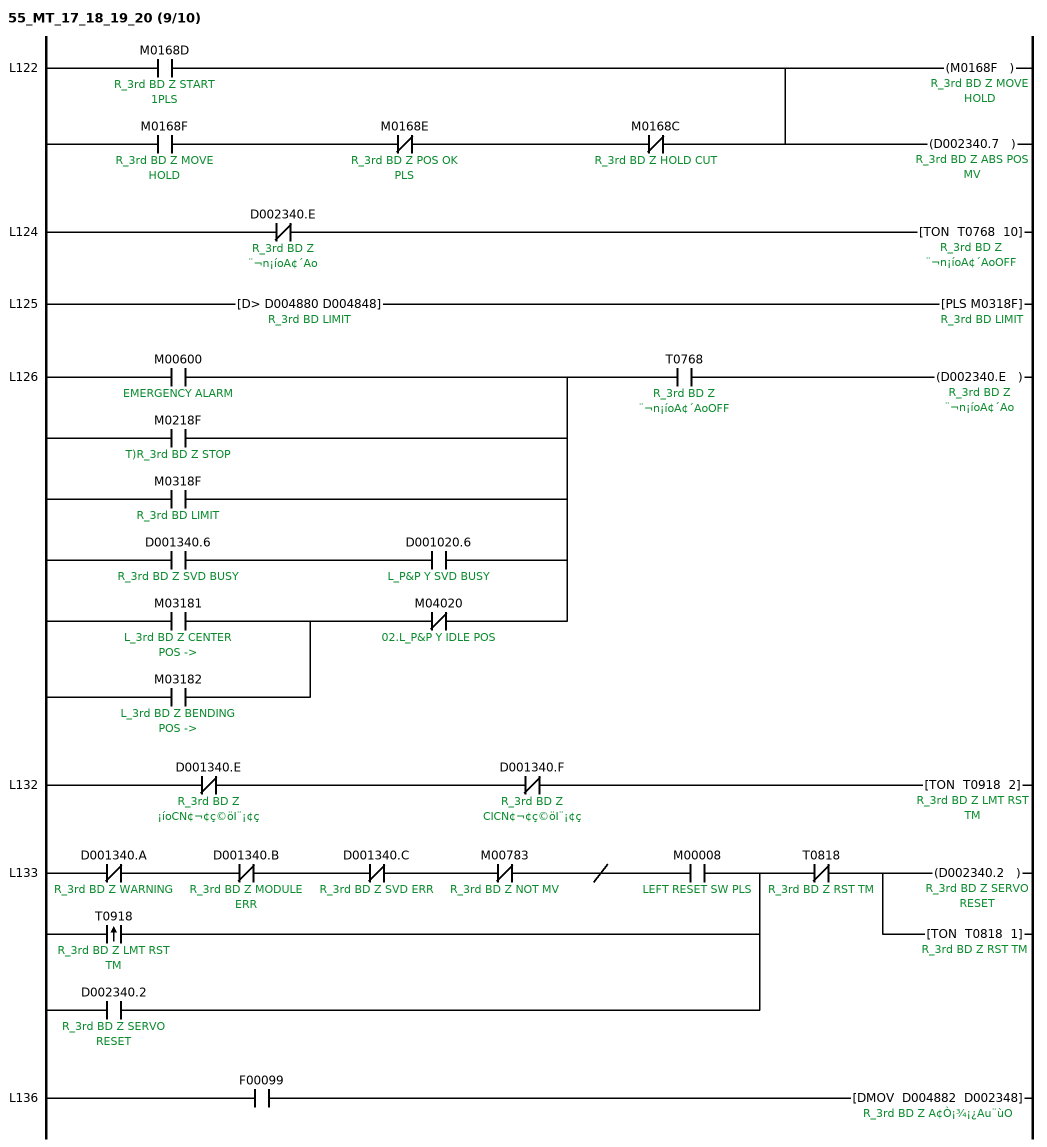
; L122
LOAD      M0168D	// R_3rd BD Z START 1PLS
LOAD      M0168F	// R_3rd BD Z MOVE HOLD
AND NOT   M0168E	// R_3rd BD Z POS OK PLS
AND NOT   M0168C	// R_3rd BD Z HOLD CUT
OR LOAD
OUT       M0168F	// R_3rd BD Z MOVE HOLD
OUT       D002340.7	// R_3rd BD Z ABS POS MV
; L124
LOAD NOT  D002340.E	// R_3rd BD Z ¨¬n¡íoA¢´Ao
TON       T0768 10	// R_3rd BD Z ¨¬n¡íoA¢´AoOFF
; L125
LOADD>    D004880 D004848	// R_3rd BD LIMIT
OUTP      M0318F	// R_3rd BD LIMIT
; L126
LOAD      M00600	// EMERGENCY ALARM
OR        M0218F	// T)R_3rd BD Z STOP
OR        M0318F	// R_3rd BD LIMIT
LOAD      D001340.6	// R_3rd BD Z SVD BUSY
AND       D001020.6	// L_P&P Y SVD BUSY
OR LOAD
LOAD      M03181	// L_3rd BD Z CENTER POS ->
OR        M03182	// L_3rd BD Z BENDING POS ->
AND NOT   M04020	// 02.L_P&P Y IDLE POS
OR LOAD
AND       T0768	// R_3rd BD Z ¨¬n¡íoA¢´AoOFF
OUT       D002340.E	// R_3rd BD Z ¨¬n¡íoA¢´Ao
; L132
LOAD NOT  D001340.E	// R_3rd BD Z ¡íoCN¢¬¢ç©öI¨¡¢ç
AND NOT   D001340.F	// R_3rd BD Z CICN¢¬¢ç©öI¨¡¢ç
TON       T0918 2	// R_3rd BD Z LMT RST TM
; L133
LOAD NOT  D001340.A	// R_3rd BD Z WARNING
AND NOT   D001340.B	// R_3rd BD Z MODULE ERR
AND NOT   D001340.C	// R_3rd BD Z SVD ERR
AND NOT   M00783	// R_3rd BD Z NOT MV
NOT
AND       M00008	// LEFT RESET SW PLS
ORP       T0918	// R_3rd BD Z LMT RST TM
OR        D002340.2	// R_3rd BD Z SERVO RESET
AND NOT   T0818	// R_3rd BD Z RST TM
OUT       D002340.2	// R_3rd BD Z SERVO RESET
TON       T0818 1	// R_3rd BD Z RST TM
; L136
LOAD      F00099
DMOV      D004882 D002348	// R_3rd BD Z A¢Ò¡¾¡¿Au¨ùO

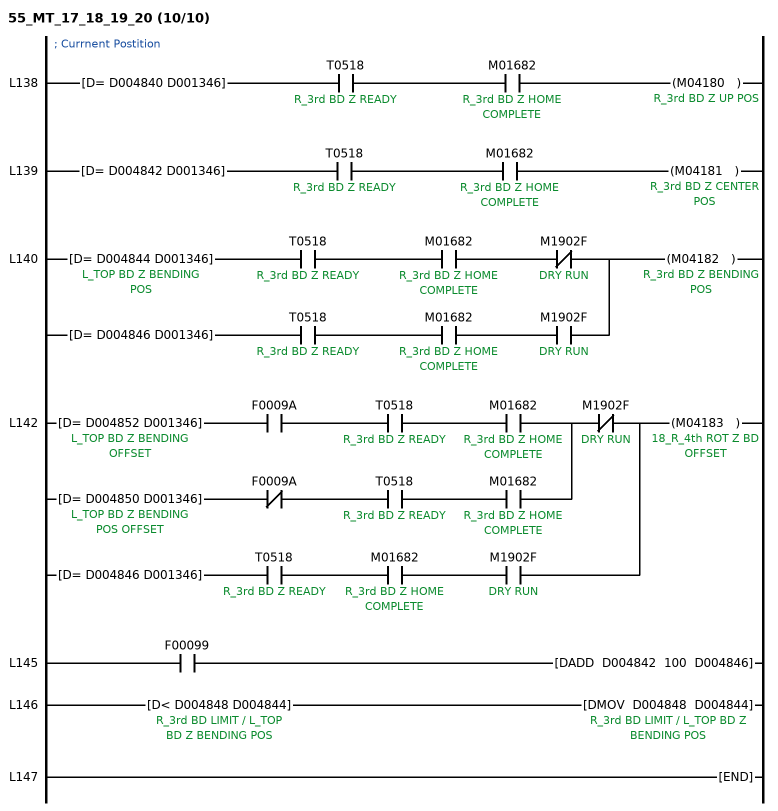
// Currnent Postition
; L138
LOADD=    D004840 D001346
AND       T0518	// R_3rd BD Z READY
AND       M01682	// R_3rd BD Z HOME COMPLETE
OUT       M04180	// R_3rd BD Z UP POS
; L139
LOADD=    D004842 D001346
AND       T0518	// R_3rd BD Z READY
AND       M01682	// R_3rd BD Z HOME COMPLETE
OUT       M04181	// R_3rd BD Z CENTER POS
; L140
LOADD=    D004844 D001346	// L_TOP BD Z BENDING POS
AND       T0518	// R_3rd BD Z READY
AND       M01682	// R_3rd BD Z HOME COMPLETE
AND NOT   M1902F	// DRY RUN
LOADD=    D004846 D001346
AND       T0518	// R_3rd BD Z READY
AND       M01682	// R_3rd BD Z HOME COMPLETE
AND       M1902F	// DRY RUN
OR LOAD
OUT       M04182	// R_3rd BD Z BENDING POS
; L142
LOADD=    D004852 D001346	// L_TOP BD Z BENDING OFFSET
AND       F0009A
AND       T0518	// R_3rd BD Z READY
AND       M01682	// R_3rd BD Z HOME COMPLETE
LOADD=    D004850 D001346	// L_TOP BD Z BENDING POS OFFSET
AND NOT   F0009A
AND       T0518	// R_3rd BD Z READY
AND       M01682	// R_3rd BD Z HOME COMPLETE
OR LOAD
AND NOT   M1902F	// DRY RUN
LOADD=    D004846 D001346
AND       T0518	// R_3rd BD Z READY
AND       M01682	// R_3rd BD Z HOME COMPLETE
AND       M1902F	// DRY RUN
OR LOAD
OUT       M04183	// 18_R_4th ROT Z BD OFFSET
; L145
LOAD      F00099
DADD      D004842 100 D004846
; L146
LOADD<    D004848 D004844	// R_3rd BD LIMIT / L_TOP BD Z BENDING POS
DMOV      D004848 D004844	// R_3rd BD LIMIT / L_TOP BD Z BENDING POS
; L147
END

PROGRAM 81_OUTPUT (task: ¨ö¨¬A¥ì CA¡¤I¡¾¡¿¡¤¡Í)

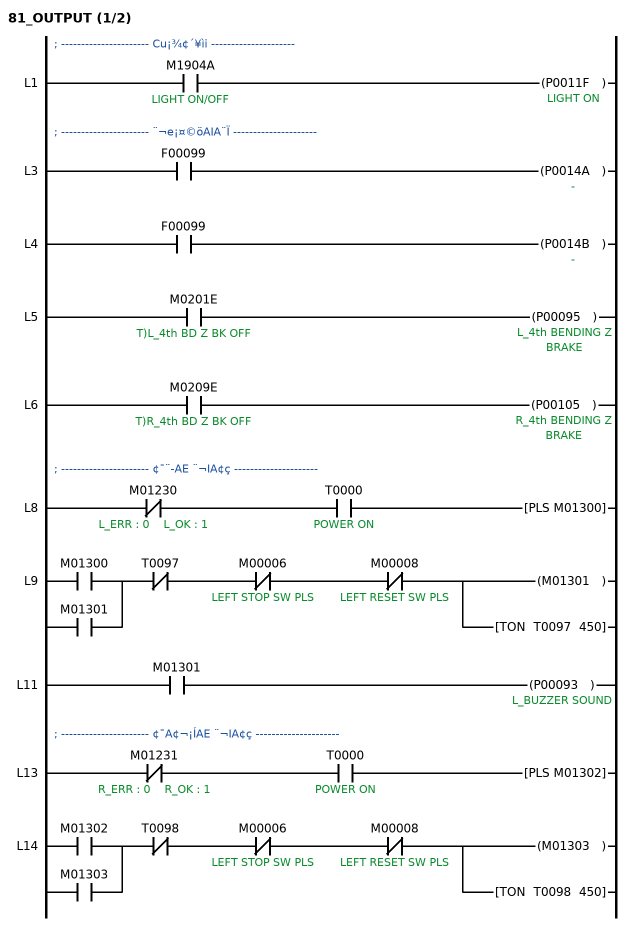
// ---------------------- Cu¡¾¢´¥ìi ---------------------
; L1
LOAD      M1904A	// LIGHT ON/OFF
OUT       P0011F	// LIGHT ON
// ---------------------- ¨¬e¡¤©öAIA¨Ï ---------------------
; L3
LOAD      F00099
OUT       P0014A	// -
; L4
LOAD      F00099
OUT       P0014B	// -
; L5
LOAD      M0201E	// T)L_4th BD Z BK OFF
OUT       P00095	// L_4th BENDING Z BRAKE
; L6
LOAD      M0209E	// T)R_4th BD Z BK OFF
OUT       P00105	// R_4th BENDING Z BRAKE
// ---------------------- ¢¯¨­AE ¨¬IA¢ç ---------------------
; L8
LOAD NOT  M01230	// L_ERR : 0    L_OK : 1
AND       T0000	// POWER ON
OUTP      M01300
; L9
LOAD      M01300
OR        M01301
AND NOT   T0097
AND NOT   M00006	// LEFT STOP SW PLS
AND NOT   M00008	// LEFT RESET SW PLS
OUT       M01301
TON       T0097 450
; L11
LOAD      M01301
OUT       P00093	// L_BUZZER SOUND
// ---------------------- ¢¯A¢¬¡ÍAE ¨¬IA¢ç ---------------------
; L13
LOAD NOT  M01231	// R_ERR : 0    R_OK : 1
AND       T0000	// POWER ON
OUTP      M01302
; L14
LOAD      M01302
OR        M01303
AND NOT   T0098
AND NOT   M00006	// LEFT STOP SW PLS
AND NOT   M00008	// LEFT RESET SW PLS
OUT       M01303
TON       T0098 450

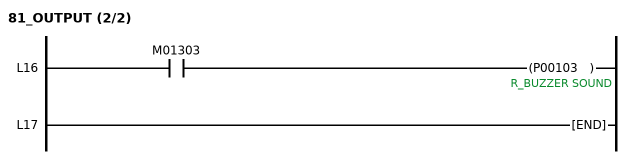
; L16
LOAD      M01303
OUT       P00103	// R_BUZZER SOUND
; L17
END

PROGRAM 82_L_MANUAL (task: ¨ö¨¬A¥ì CA¡¤I¡¾¡¿¡¤¡Í)

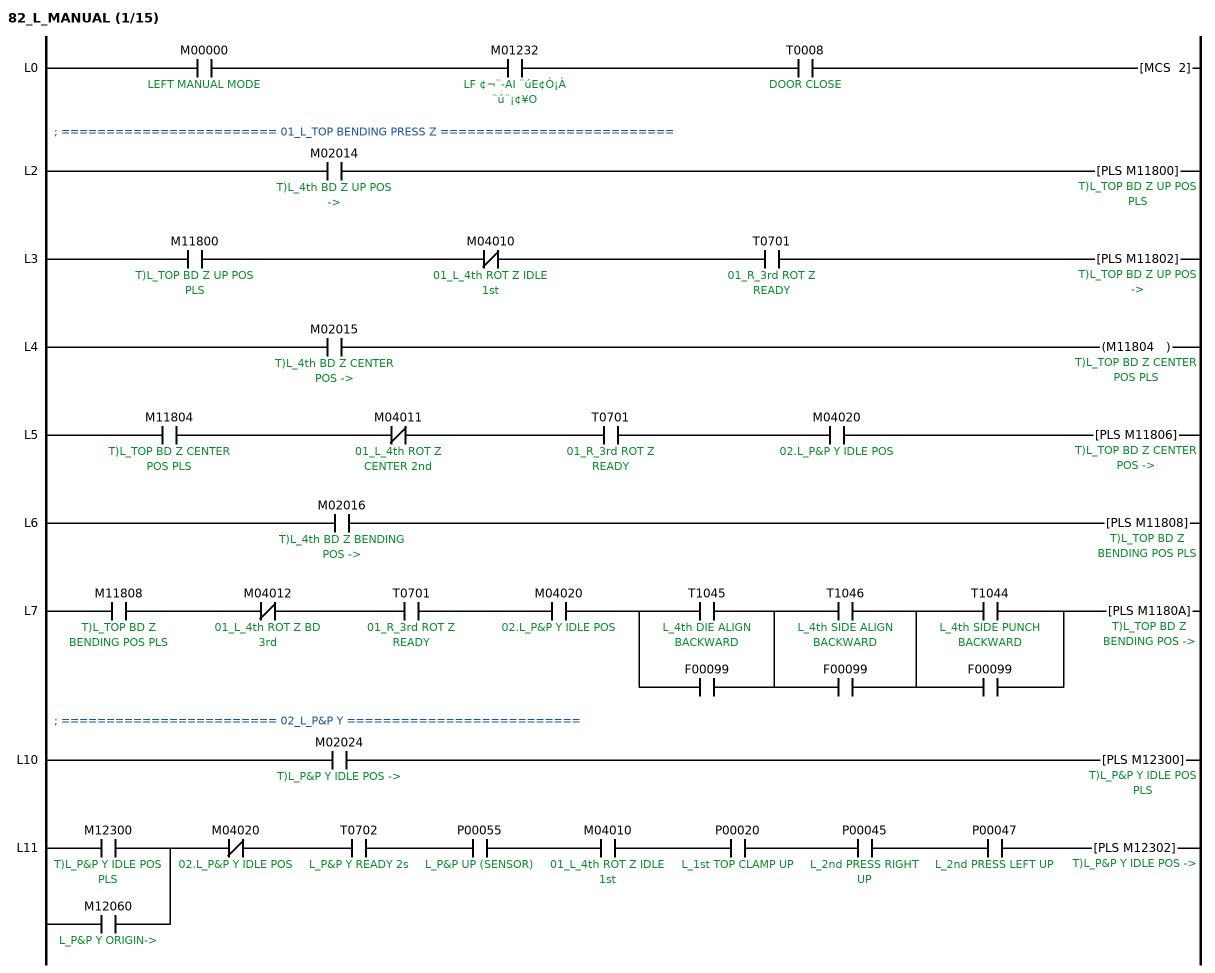
; L0
LOAD      M00000	// LEFT MANUAL MODE
AND       M01232	// LF ¢¬¨­AI ¨úE¢Ò¡À ¨ú¨¡¢¥O
AND       T0008	// DOOR CLOSE
MCS       2
// ======================== 01_L_TOP BENDING PRESS Z ==========================
; L2
LOAD      M02014	// T)L_4th BD Z UP POS ->
OUTP      M11800	// T)L_TOP BD Z UP POS PLS
; L3
LOAD      M11800	// T)L_TOP BD Z UP POS PLS
AND NOT   M04010	// 01_L_4th ROT Z IDLE 1st
AND       T0701	// 01_R_3rd ROT Z READY
OUTP      M11802	// T)L_TOP BD Z UP POS ->
; L4
LOAD      M02015	// T)L_4th BD Z CENTER POS ->
OUT       M11804	// T)L_TOP BD Z CENTER POS PLS
; L5
LOAD      M11804	// T)L_TOP BD Z CENTER POS PLS
AND NOT   M04011	// 01_L_4th ROT Z CENTER 2nd
AND       T0701	// 01_R_3rd ROT Z READY
AND       M04020	// 02.L_P&P Y IDLE POS
OUTP      M11806	// T)L_TOP BD Z CENTER POS ->
; L6
LOAD      M02016	// T)L_4th BD Z BENDING POS ->
OUTP      M11808	// T)L_TOP BD Z BENDING POS PLS
; L7
LOAD      M11808	// T)L_TOP BD Z BENDING POS PLS
AND NOT   M04012	// 01_L_4th ROT Z BD 3rd
AND       T0701	// 01_R_3rd ROT Z READY
AND       M04020	// 02.L_P&P Y IDLE POS
LOAD      T1045	// L_4th DIE ALIGN BACKWARD
OR        F00099
AND LOAD
LOAD      T1046	// L_4th SIDE ALIGN BACKWARD
OR        F00099
AND LOAD
LOAD      T1044	// L_4th SIDE PUNCH BACKWARD
OR        F00099
AND LOAD
OUTP      M1180A	// T)L_TOP BD Z BENDING POS ->
// ======================== 02_L_P&P Y ==========================
; L10
LOAD      M02024	// T)L_P&P Y IDLE POS ->
OUTP      M12300	// T)L_P&P Y IDLE POS PLS
; L11
LOAD      M12300	// T)L_P&P Y IDLE POS PLS
OR        M12060	// L_P&P Y ORIGIN->
AND NOT   M04020	// 02.L_P&P Y IDLE POS
AND       T0702	// L_P&P Y READY 2s
AND       P00055	// L_P&P UP (SENSOR)
AND       M04010	// 01_L_4th ROT Z IDLE 1st
AND       P00020	// L_1st TOP CLAMP UP
AND       P00045	// L_2nd PRESS RIGHT UP
AND       P00047	// L_2nd PRESS LEFT UP
OUTP      M12302	// T)L_P&P Y IDLE POS ->

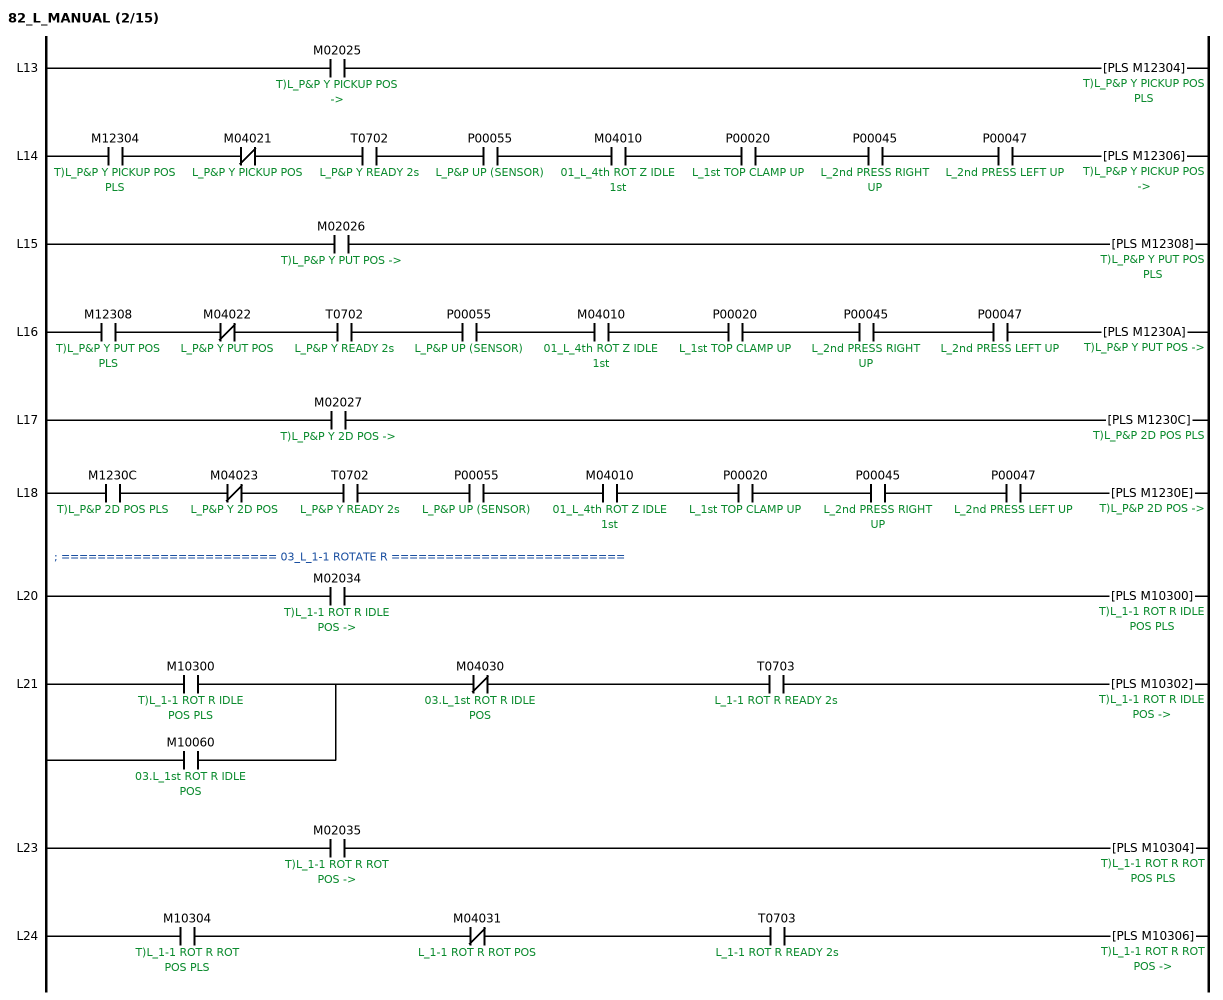
; L13
LOAD      M02025	// T)L_P&P Y PICKUP POS ->
OUTP      M12304	// T)L_P&P Y PICKUP POS PLS
; L14
LOAD      M12304	// T)L_P&P Y PICKUP POS PLS
AND NOT   M04021	// L_P&P Y PICKUP POS
AND       T0702	// L_P&P Y READY 2s
AND       P00055	// L_P&P UP (SENSOR)
AND       M04010	// 01_L_4th ROT Z IDLE 1st
AND       P00020	// L_1st TOP CLAMP UP
AND       P00045	// L_2nd PRESS RIGHT UP
AND       P00047	// L_2nd PRESS LEFT UP
OUTP      M12306	// T)L_P&P Y PICKUP POS ->
; L15
LOAD      M02026	// T)L_P&P Y PUT POS ->
OUTP      M12308	// T)L_P&P Y PUT POS PLS
; L16
LOAD      M12308	// T)L_P&P Y PUT POS PLS
AND NOT   M04022	// L_P&P Y PUT POS
AND       T0702	// L_P&P Y READY 2s
AND       P00055	// L_P&P UP (SENSOR)
AND       M04010	// 01_L_4th ROT Z IDLE 1st
AND       P00020	// L_1st TOP CLAMP UP
AND       P00045	// L_2nd PRESS RIGHT UP
AND       P00047	// L_2nd PRESS LEFT UP
OUTP      M1230A	// T)L_P&P Y PUT POS ->
; L17
LOAD      M02027	// T)L_P&P Y 2D POS ->
OUTP      M1230C	// T)L_P&P 2D POS PLS
; L18
LOAD      M1230C	// T)L_P&P 2D POS PLS
AND NOT   M04023	// L_P&P Y 2D POS
AND       T0702	// L_P&P Y READY 2s
AND       P00055	// L_P&P UP (SENSOR)
AND       M04010	// 01_L_4th ROT Z IDLE 1st
AND       P00020	// L_1st TOP CLAMP UP
AND       P00045	// L_2nd PRESS RIGHT UP
AND       P00047	// L_2nd PRESS LEFT UP
OUTP      M1230E	// T)L_P&P 2D POS ->
// ======================== 03_L_1-1 ROTATE R ==========================
; L20
LOAD      M02034	// T)L_1-1 ROT R IDLE POS ->
OUTP      M10300	// T)L_1-1 ROT R IDLE POS PLS
; L21
LOAD      M10300	// T)L_1-1 ROT R IDLE POS PLS
OR        M10060	// 03.L_1st ROT R IDLE POS
AND NOT   M04030	// 03.L_1st ROT R IDLE POS
AND       T0703	// L_1-1 ROT R READY 2s
OUTP      M10302	// T)L_1-1 ROT R IDLE POS ->
; L23
LOAD      M02035	// T)L_1-1 ROT R ROT POS ->
OUTP      M10304	// T)L_1-1 ROT R ROT POS PLS
; L24
LOAD      M10304	// T)L_1-1 ROT R ROT POS PLS
AND NOT   M04031	// L_1-1 ROT R ROT POS
AND       T0703	// L_1-1 ROT R READY 2s
OUTP      M10306	// T)L_1-1 ROT R ROT POS ->

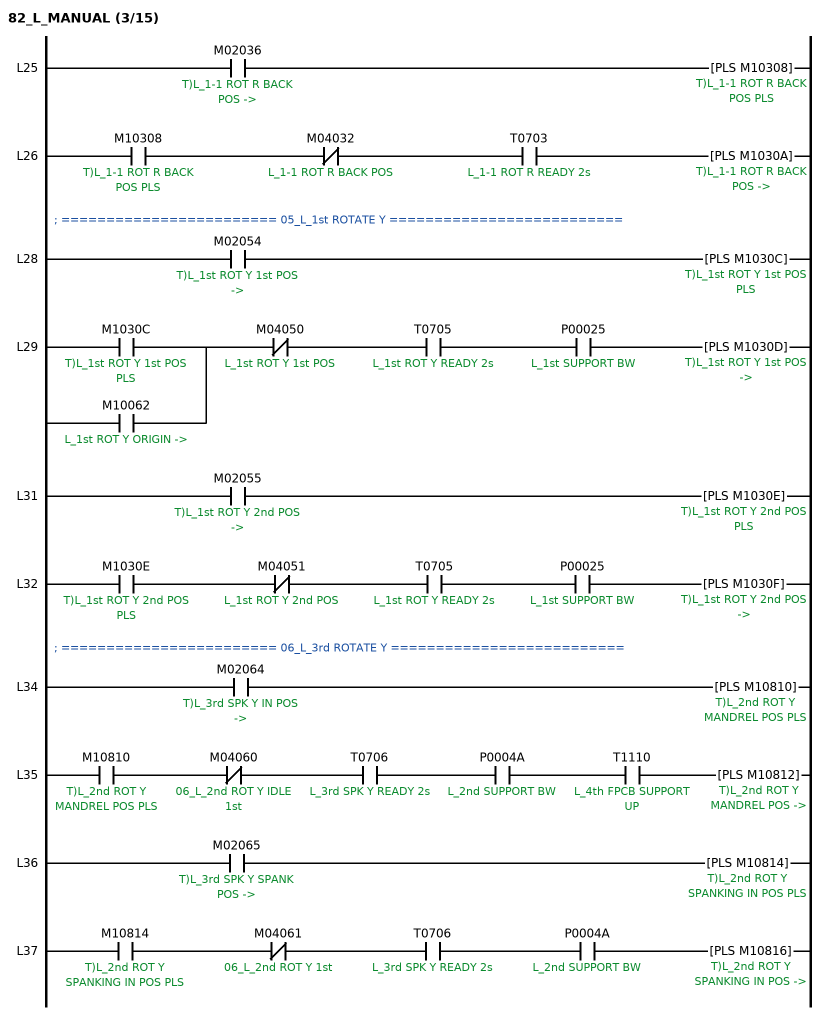
; L25
LOAD      M02036	// T)L_1-1 ROT R BACK POS ->
OUTP      M10308	// T)L_1-1 ROT R BACK POS PLS
; L26
LOAD      M10308	// T)L_1-1 ROT R BACK POS PLS
AND NOT   M04032	// L_1-1 ROT R BACK POS
AND       T0703	// L_1-1 ROT R READY 2s
OUTP      M1030A	// T)L_1-1 ROT R BACK POS ->
// ======================== 05_L_1st ROTATE Y ==========================
; L28
LOAD      M02054	// T)L_1st ROT Y 1st POS ->
OUTP      M1030C	// T)L_1st ROT Y 1st POS PLS
; L29
LOAD      M1030C	// T)L_1st ROT Y 1st POS PLS
OR        M10062	// L_1st ROT Y ORIGIN ->
AND NOT   M04050	// L_1st ROT Y 1st POS
AND       T0705	// L_1st ROT Y READY 2s
AND       P00025	// L_1st SUPPORT BW
OUTP      M1030D	// T)L_1st ROT Y 1st POS ->
; L31
LOAD      M02055	// T)L_1st ROT Y 2nd POS ->
OUTP      M1030E	// T)L_1st ROT Y 2nd POS PLS
; L32
LOAD      M1030E	// T)L_1st ROT Y 2nd POS PLS
AND NOT   M04051	// L_1st ROT Y 2nd POS
AND       T0705	// L_1st ROT Y READY 2s
AND       P00025	// L_1st SUPPORT BW
OUTP      M1030F	// T)L_1st ROT Y 2nd POS ->
// ======================== 06_L_3rd ROTATE Y ==========================
; L34
LOAD      M02064	// T)L_3rd SPK Y IN POS ->
OUTP      M10810	// T)L_2nd ROT Y MANDREL POS PLS
; L35
LOAD      M10810	// T)L_2nd ROT Y MANDREL POS PLS
AND NOT   M04060	// 06_L_2nd ROT Y IDLE 1st
AND       T0706	// L_3rd SPK Y READY 2s
AND       P0004A	// L_2nd SUPPORT BW
AND       T1110	// L_4th FPCB SUPPORT UP
OUTP      M10812	// T)L_2nd ROT Y MANDREL POS ->
; L36
LOAD      M02065	// T)L_3rd SPK Y SPANK POS ->
OUTP      M10814	// T)L_2nd ROT Y SPANKING IN POS PLS
; L37
LOAD      M10814	// T)L_2nd ROT Y SPANKING IN POS PLS
AND NOT   M04061	// 06_L_2nd ROT Y 1st
AND       T0706	// L_3rd SPK Y READY 2s
AND       P0004A	// L_2nd SUPPORT BW
OUTP      M10816	// T)L_2nd ROT Y SPANKING IN POS ->

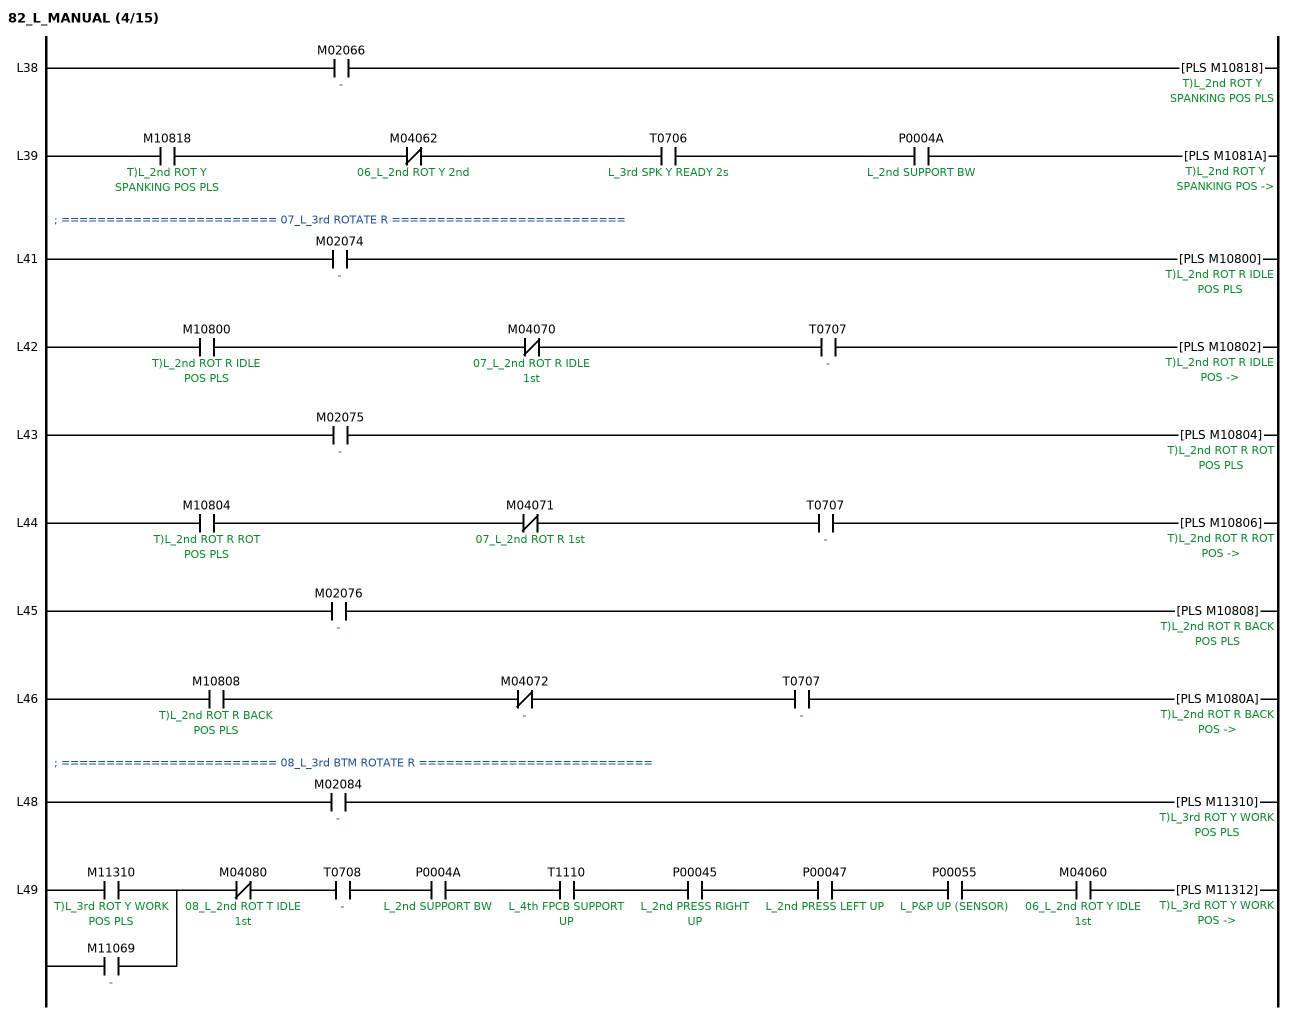
; L38
LOAD      M02066	// -
OUTP      M10818	// T)L_2nd ROT Y SPANKING POS PLS
; L39
LOAD      M10818	// T)L_2nd ROT Y SPANKING POS PLS
AND NOT   M04062	// 06_L_2nd ROT Y 2nd
AND       T0706	// L_3rd SPK Y READY 2s
AND       P0004A	// L_2nd SUPPORT BW
OUTP      M1081A	// T)L_2nd ROT Y SPANKING POS ->
// ======================== 07_L_3rd ROTATE R ==========================
; L41
LOAD      M02074	// -
OUTP      M10800	// T)L_2nd ROT R IDLE POS PLS
; L42
LOAD      M10800	// T)L_2nd ROT R IDLE POS PLS
AND NOT   M04070	// 07_L_2nd ROT R IDLE 1st
AND       T0707	// -
OUTP      M10802	// T)L_2nd ROT R IDLE POS ->
; L43
LOAD      M02075	// -
OUTP      M10804	// T)L_2nd ROT R ROT POS PLS
; L44
LOAD      M10804	// T)L_2nd ROT R ROT POS PLS
AND NOT   M04071	// 07_L_2nd ROT R 1st
AND       T0707	// -
OUTP      M10806	// T)L_2nd ROT R ROT POS ->
; L45
LOAD      M02076	// -
OUTP      M10808	// T)L_2nd ROT R BACK POS PLS
; L46
LOAD      M10808	// T)L_2nd ROT R BACK POS PLS
AND NOT   M04072	// -
AND       T0707	// -
OUTP      M1080A	// T)L_2nd ROT R BACK POS ->
// ======================== 08_L_3rd BTM ROTATE R ==========================
; L48
LOAD      M02084	// -
OUTP      M11310	// T)L_3rd ROT Y WORK POS PLS
; L49
LOAD      M11310	// T)L_3rd ROT Y WORK POS PLS
OR        M11069	// -
AND NOT   M04080	// 08_L_2nd ROT T IDLE 1st
AND       T0708	// -
AND       P0004A	// L_2nd SUPPORT BW
AND       T1110	// L_4th FPCB SUPPORT UP
AND       P00045	// L_2nd PRESS RIGHT UP
AND       P00047	// L_2nd PRESS LEFT UP
AND       P00055	// L_P&P UP (SENSOR)
AND       M04060	// 06_L_2nd ROT Y IDLE 1st
OUTP      M11312	// T)L_3rd ROT Y WORK POS ->

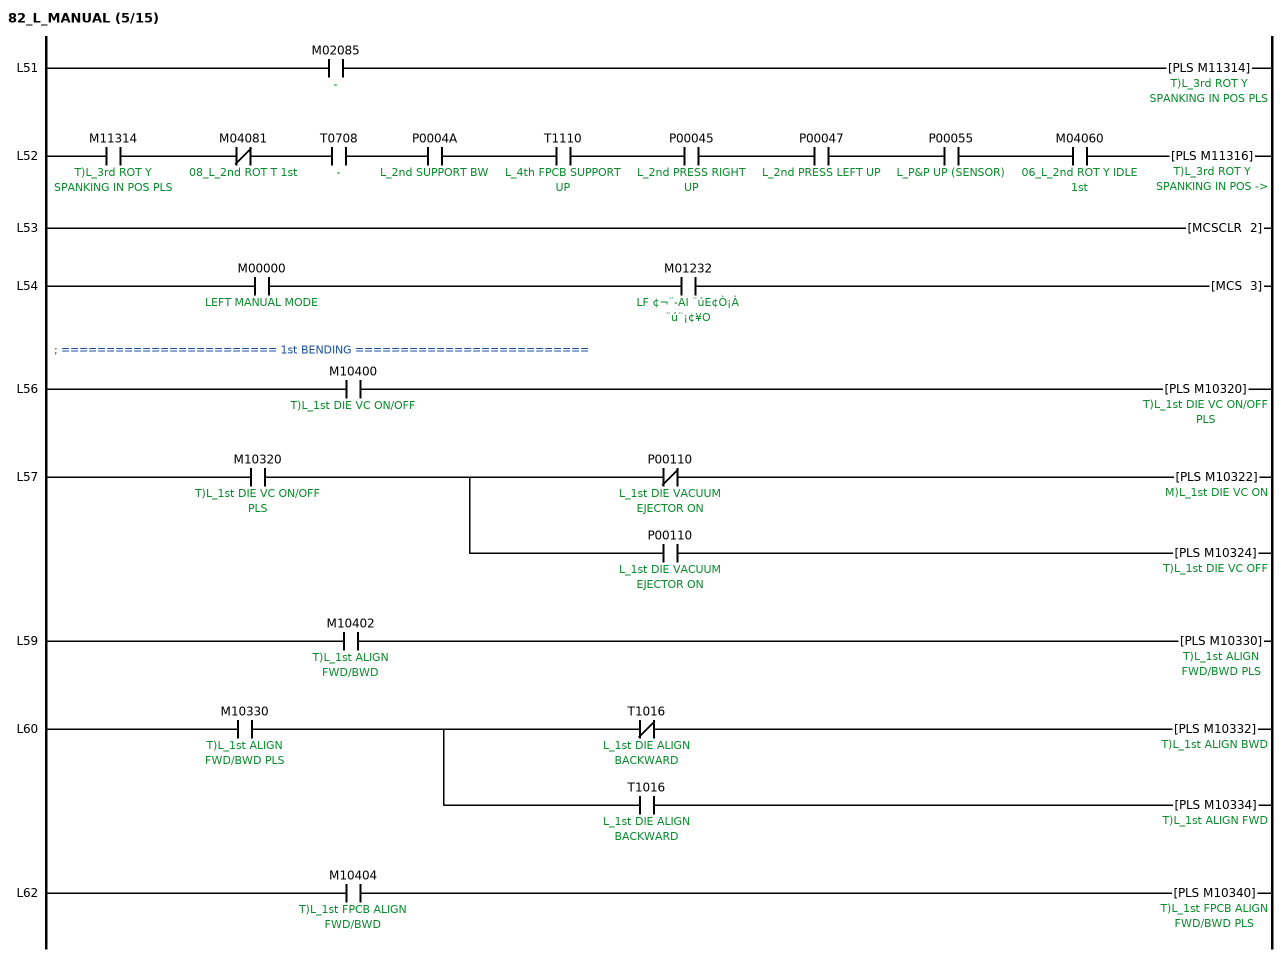
; L51
LOAD      M02085	// -
OUTP      M11314	// T)L_3rd ROT Y SPANKING IN POS PLS
; L52
LOAD      M11314	// T)L_3rd ROT Y SPANKING IN POS PLS
AND NOT   M04081	// 08_L_2nd ROT T 1st
AND       T0708	// -
AND       P0004A	// L_2nd SUPPORT BW
AND       T1110	// L_4th FPCB SUPPORT UP
AND       P00045	// L_2nd PRESS RIGHT UP
AND       P00047	// L_2nd PRESS LEFT UP
AND       P00055	// L_P&P UP (SENSOR)
AND       M04060	// 06_L_2nd ROT Y IDLE 1st
OUTP      M11316	// T)L_3rd ROT Y SPANKING IN POS ->
; L53
MCSCLR    2
; L54
LOAD      M00000	// LEFT MANUAL MODE
AND       M01232	// LF ¢¬¨­AI ¨úE¢Ò¡À ¨ú¨¡¢¥O
MCS       3
// ======================== 1st BENDING ==========================
; L56
LOAD      M10400	// T)L_1st DIE VC ON/OFF
OUTP      M10320	// T)L_1st DIE VC ON/OFF PLS
; L57
LOAD      M10320	// T)L_1st DIE VC ON/OFF PLS
MPUSH
AND NOT   P00110	// L_1st DIE VACUUM EJECTOR ON
OUTP      M10322	// M)L_1st DIE VC ON
MPOP
AND       P00110	// L_1st DIE VACUUM EJECTOR ON
OUTP      M10324	// T)L_1st DIE VC OFF
; L59
LOAD      M10402	// T)L_1st ALIGN FWD/BWD
OUTP      M10330	// T)L_1st ALIGN FWD/BWD PLS
; L60
LOAD      M10330	// T)L_1st ALIGN FWD/BWD PLS
MPUSH
AND NOT   T1016	// L_1st DIE ALIGN BACKWARD
OUTP      M10332	// T)L_1st ALIGN BWD
MPOP
AND       T1016	// L_1st DIE ALIGN BACKWARD
OUTP      M10334	// T)L_1st ALIGN FWD
; L62
LOAD      M10404	// T)L_1st FPCB ALIGN FWD/BWD
OUTP      M10340	// T)L_1st FPCB ALIGN FWD/BWD PLS

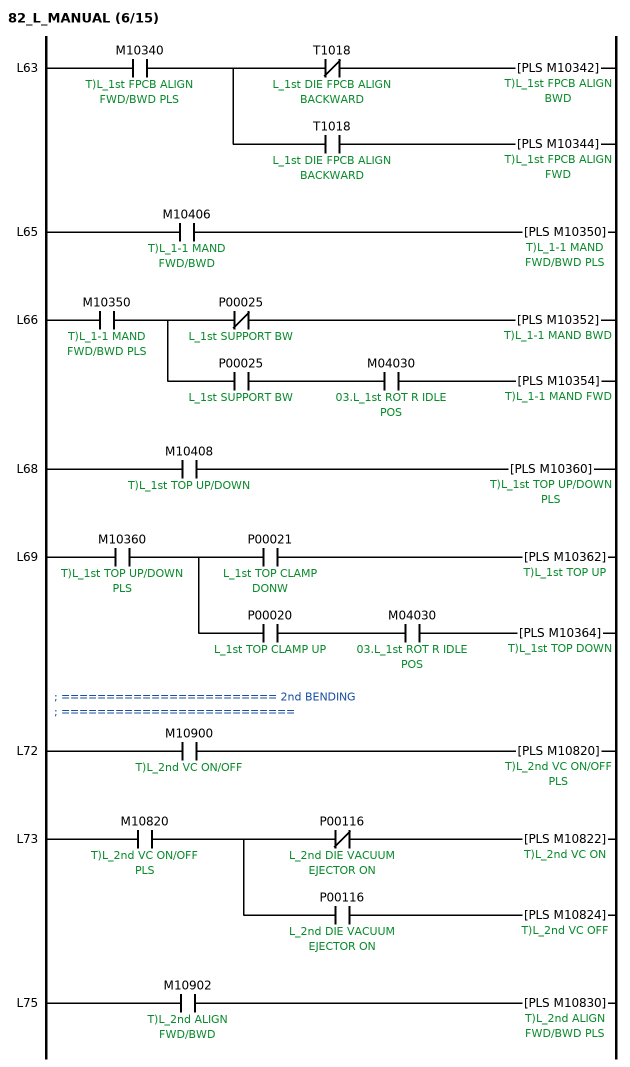
; L63
LOAD      M10340	// T)L_1st FPCB ALIGN FWD/BWD PLS
MPUSH
AND NOT   T1018	// L_1st DIE FPCB ALIGN BACKWARD
OUTP      M10342	// T)L_1st FPCB ALIGN BWD
MPOP
AND       T1018	// L_1st DIE FPCB ALIGN BACKWARD
OUTP      M10344	// T)L_1st FPCB ALIGN FWD
; L65
LOAD      M10406	// T)L_1-1 MAND FWD/BWD
OUTP      M10350	// T)L_1-1 MAND FWD/BWD PLS
; L66
LOAD      M10350	// T)L_1-1 MAND FWD/BWD PLS
MPUSH
AND NOT   P00025	// L_1st SUPPORT BW
OUTP      M10352	// T)L_1-1 MAND BWD
MPOP
AND       P00025	// L_1st SUPPORT BW
AND       M04030	// 03.L_1st ROT R IDLE POS
OUTP      M10354	// T)L_1-1 MAND FWD
; L68
LOAD      M10408	// T)L_1st TOP UP/DOWN
OUTP      M10360	// T)L_1st TOP UP/DOWN PLS
; L69
LOAD      M10360	// T)L_1st TOP UP/DOWN PLS
MPUSH
AND       P00021	// L_1st TOP CLAMP DONW
OUTP      M10362	// T)L_1st TOP UP
MPOP
AND       P00020	// L_1st TOP CLAMP UP
AND       M04030	// 03.L_1st ROT R IDLE POS
OUTP      M10364	// T)L_1st TOP DOWN
// ======================== 2nd BENDING ==========================
; L72
LOAD      M10900	// T)L_2nd VC ON/OFF
OUTP      M10820	// T)L_2nd VC ON/OFF PLS
; L73
LOAD      M10820	// T)L_2nd VC ON/OFF PLS
MPUSH
AND NOT   P00116	// L_2nd DIE VACUUM EJECTOR ON
OUTP      M10822	// T)L_2nd VC ON
MPOP
AND       P00116	// L_2nd DIE VACUUM EJECTOR ON
OUTP      M10824	// T)L_2nd VC OFF
; L75
LOAD      M10902	// T)L_2nd ALIGN FWD/BWD
OUTP      M10830	// T)L_2nd ALIGN FWD/BWD PLS

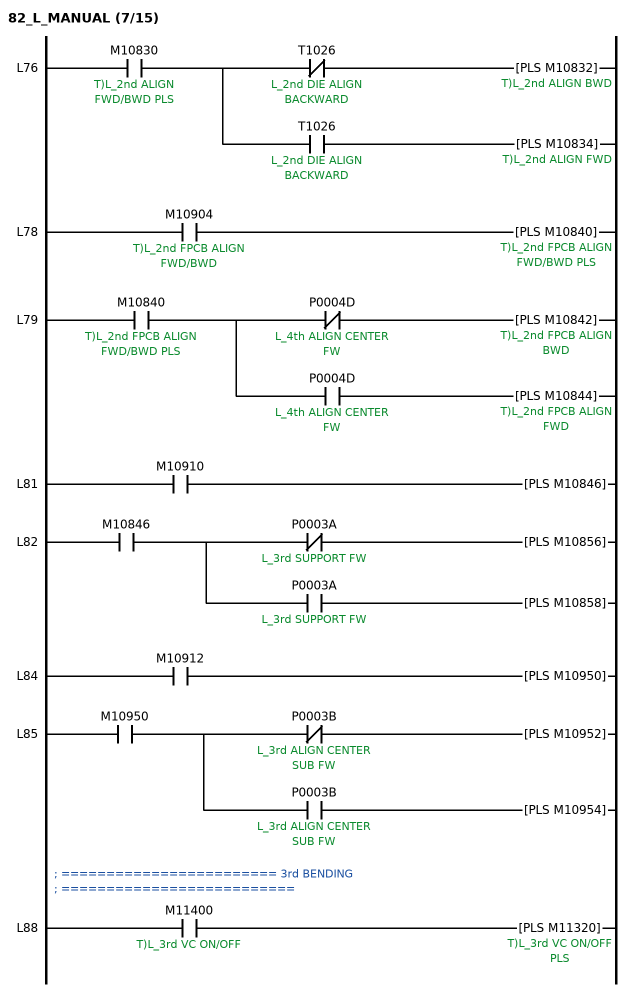
; L76
LOAD      M10830	// T)L_2nd ALIGN FWD/BWD PLS
MPUSH
AND NOT   T1026	// L_2nd DIE ALIGN BACKWARD
OUTP      M10832	// T)L_2nd ALIGN BWD
MPOP
AND       T1026	// L_2nd DIE ALIGN BACKWARD
OUTP      M10834	// T)L_2nd ALIGN FWD
; L78
LOAD      M10904	// T)L_2nd FPCB ALIGN FWD/BWD
OUTP      M10840	// T)L_2nd FPCB ALIGN FWD/BWD PLS
; L79
LOAD      M10840	// T)L_2nd FPCB ALIGN FWD/BWD PLS
MPUSH
AND NOT   P0004D	// L_4th ALIGN CENTER FW
OUTP      M10842	// T)L_2nd FPCB ALIGN BWD
MPOP
AND       P0004D	// L_4th ALIGN CENTER FW
OUTP      M10844	// T)L_2nd FPCB ALIGN FWD
; L81
LOAD      M10910
OUTP      M10846
; L82
LOAD      M10846
MPUSH
AND NOT   P0003A	// L_3rd SUPPORT FW
OUTP      M10856
MPOP
AND       P0003A	// L_3rd SUPPORT FW
OUTP      M10858
; L84
LOAD      M10912
OUTP      M10950
; L85
LOAD      M10950
MPUSH
AND NOT   P0003B	// L_3rd ALIGN CENTER SUB FW
OUTP      M10952
MPOP
AND       P0003B	// L_3rd ALIGN CENTER SUB FW
OUTP      M10954
// ======================== 3rd BENDING ==========================
; L88
LOAD      M11400	// T)L_3rd VC ON/OFF
OUTP      M11320	// T)L_3rd VC ON/OFF PLS

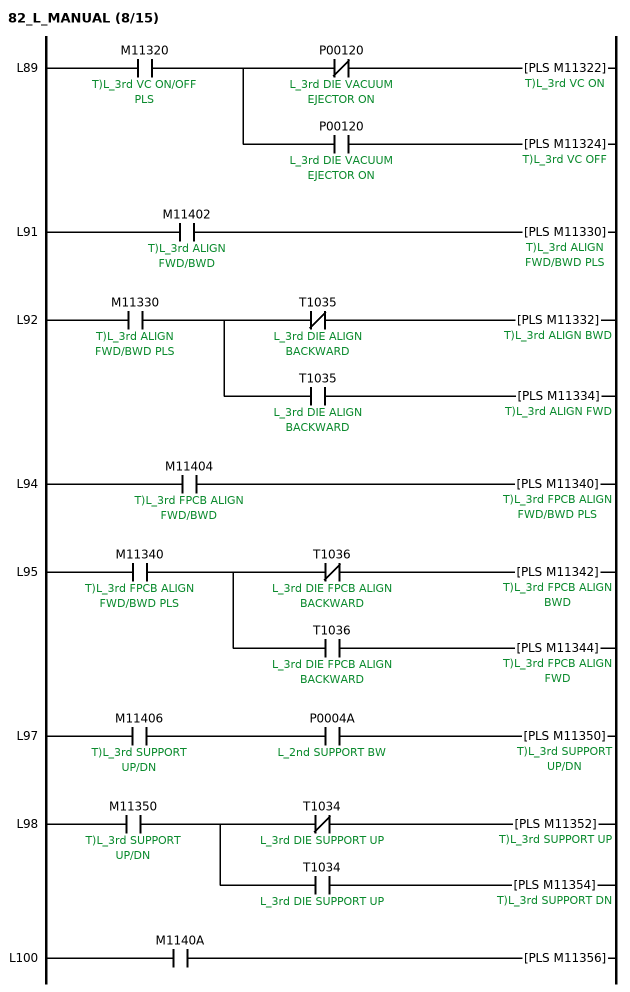
; L89
LOAD      M11320	// T)L_3rd VC ON/OFF PLS
MPUSH
AND NOT   P00120	// L_3rd DIE VACUUM EJECTOR ON
OUTP      M11322	// T)L_3rd VC ON
MPOP
AND       P00120	// L_3rd DIE VACUUM EJECTOR ON
OUTP      M11324	// T)L_3rd VC OFF
; L91
LOAD      M11402	// T)L_3rd ALIGN FWD/BWD
OUTP      M11330	// T)L_3rd ALIGN FWD/BWD PLS
; L92
LOAD      M11330	// T)L_3rd ALIGN FWD/BWD PLS
MPUSH
AND NOT   T1035	// L_3rd DIE ALIGN BACKWARD
OUTP      M11332	// T)L_3rd ALIGN BWD
MPOP
AND       T1035	// L_3rd DIE ALIGN BACKWARD
OUTP      M11334	// T)L_3rd ALIGN FWD
; L94
LOAD      M11404	// T)L_3rd FPCB ALIGN FWD/BWD
OUTP      M11340	// T)L_3rd FPCB ALIGN FWD/BWD PLS
; L95
LOAD      M11340	// T)L_3rd FPCB ALIGN FWD/BWD PLS
MPUSH
AND NOT   T1036	// L_3rd DIE FPCB ALIGN BACKWARD
OUTP      M11342	// T)L_3rd FPCB ALIGN BWD
MPOP
AND       T1036	// L_3rd DIE FPCB ALIGN BACKWARD
OUTP      M11344	// T)L_3rd FPCB ALIGN FWD
; L97
LOAD      M11406	// T)L_3rd SUPPORT UP/DN
AND       P0004A	// L_2nd SUPPORT BW
OUTP      M11350	// T)L_3rd SUPPORT UP/DN
; L98
LOAD      M11350	// T)L_3rd SUPPORT UP/DN
MPUSH
AND NOT   T1034	// L_3rd DIE SUPPORT UP
OUTP      M11352	// T)L_3rd SUPPORT UP
MPOP
AND       T1034	// L_3rd DIE SUPPORT UP
OUTP      M11354	// T)L_3rd SUPPORT DN
; L100
LOAD      M1140A
OUTP      M11356

